Yaskawa INFORM job: A_ROOF_UPPER_0614_2_PAINT_19.JBI

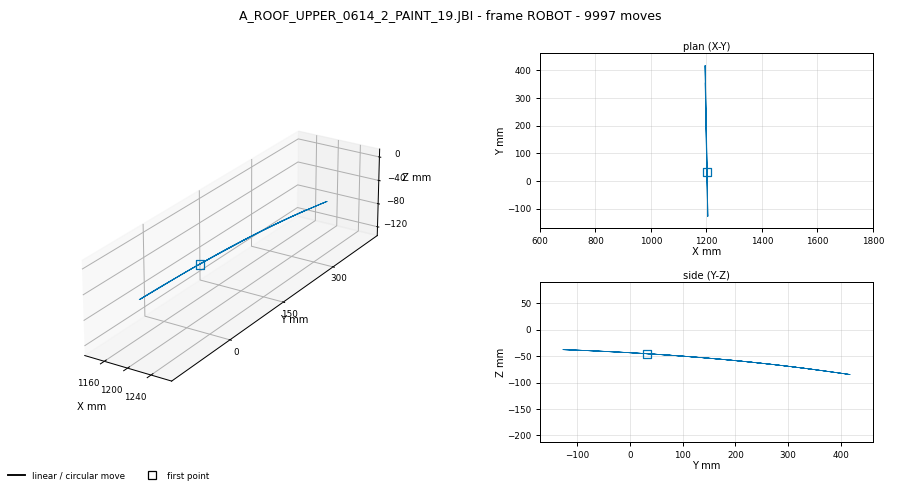
[picture p0: tool path of A_ROOF_UPPER_0614_2_PAINT_19.JBI in frame ROBOT, 9997 of 9997 moves have a stored position in this frame; points joined in program order, loops and branches not executed]
/JOB
//NAME A_ROOF_UPPER_0614_2_PAINT19
//POS
///NPOS 9997,0,0,0,0,0
///TOOL 1
///USER 0
///POSTYPE ROBOT
///RECTAN
///RCONF 1,0,0,0,0,0,0,0,0,0,0,0,0,0,0,0,0,0,0,0,0,0,0,0
C00000=1202.977,32.541,-45.099,-179.409,5.654,148.820
C00001=1202.972,32.790,-45.114,-179.406,5.654,148.820
C00002=1202.968,33.040,-45.130,-179.403,5.655,148.819
C00003=1202.962,33.290,-45.145,-179.401,5.655,148.818
C00004=1202.958,33.539,-45.160,-179.399,5.656,148.818
C00005=1202.952,33.788,-45.176,-179.396,5.657,148.817
C00006=1202.948,34.037,-45.191,-179.393,5.657,148.817
C00007=1202.943,34.287,-45.207,-179.391,5.658,148.816
C00008=1202.937,34.537,-45.222,-179.388,5.658,148.815
C00009=1202.933,34.786,-45.237,-179.386,5.659,148.815
C00010=1202.927,35.035,-45.253,-179.383,5.660,148.814
C00011=1202.923,35.285,-45.269,-179.380,5.660,148.813
C00012=1202.917,35.535,-45.285,-179.378,5.661,148.813
C00013=1202.912,35.784,-45.300,-179.376,5.661,148.812
C00014=1202.907,36.033,-45.315,-179.373,5.662,148.812
C00015=1202.902,36.283,-45.331,-179.370,5.663,148.811
C00016=1202.898,36.532,-45.347,-179.368,5.663,148.810
C00017=1202.893,36.781,-45.362,-179.365,5.664,148.810
C00018=1202.888,37.031,-45.378,-179.363,5.664,148.809
C00019=1202.882,37.281,-45.394,-179.360,5.665,148.808
C00020=1202.878,37.530,-45.409,-179.358,5.666,148.808
C00021=1202.872,37.779,-45.425,-179.355,5.666,148.807
C00022=1202.868,38.029,-45.440,-179.353,5.667,148.807
C00023=1202.862,38.279,-45.456,-179.350,5.667,148.806
C00024=1202.858,38.528,-45.471,-179.347,5.669,148.805
C00025=1202.853,38.778,-45.487,-179.344,5.669,148.805
C00026=1202.848,39.027,-45.503,-179.342,5.670,148.804
C00027=1202.842,39.276,-45.519,-179.340,5.671,148.804
C00028=1202.838,39.526,-45.534,-179.337,5.671,148.803
C00029=1202.833,39.775,-45.550,-179.334,5.672,148.802
C00030=1202.827,40.025,-45.565,-179.332,5.672,148.802
C00031=1202.823,40.274,-45.582,-179.330,5.673,148.801
C00032=1202.818,40.523,-45.598,-179.327,5.674,148.800
C00033=1202.813,40.773,-45.613,-179.324,5.674,148.800
C00034=1202.808,41.023,-45.629,-179.322,5.675,148.799
C00035=1202.803,41.272,-45.644,-179.319,5.676,148.799
C00036=1202.798,41.521,-45.661,-179.317,5.676,148.798
C00037=1202.793,41.771,-45.676,-179.314,5.677,148.797
C00038=1202.788,42.020,-45.692,-179.312,5.677,148.797
C00039=1202.783,42.269,-45.707,-179.309,5.678,148.796
C00040=1202.778,42.519,-45.724,-179.307,5.679,148.795
C00041=1202.773,42.768,-45.739,-179.304,5.679,148.795
C00042=1202.768,43.018,-45.755,-179.301,5.680,148.794
C00043=1202.763,43.267,-45.772,-179.299,5.682,148.794
C00044=1202.758,43.517,-45.787,-179.296,5.682,148.793
C00045=1202.753,43.767,-45.803,-179.293,5.683,148.792
C00046=1202.748,44.016,-45.819,-179.291,5.683,148.792
C00047=1202.743,44.265,-45.835,-179.289,5.684,148.791
C00048=1202.738,44.515,-45.850,-179.286,5.685,148.791
C00049=1202.733,44.763,-45.867,-179.283,5.685,148.790
C00050=1202.729,45.014,-45.883,-179.281,5.686,148.789
C00051=1202.723,45.263,-45.898,-179.279,5.687,148.789
C00052=1202.719,45.512,-45.915,-179.276,5.687,148.788
C00053=1202.713,45.762,-45.930,-179.273,5.688,148.787
C00054=1202.708,46.011,-45.946,-179.271,5.688,148.787
C00055=1202.703,46.261,-45.963,-179.269,5.689,148.786
C00056=1202.698,46.510,-45.978,-179.266,5.690,148.786
C00057=1202.694,46.760,-45.995,-179.263,5.691,148.785
C00058=1202.688,47.009,-46.011,-179.260,5.691,148.784
C00059=1202.683,47.259,-46.027,-179.258,5.692,148.784
C00060=1202.678,47.508,-46.043,-179.255,5.693,148.783
C00061=1202.673,47.757,-46.058,-179.253,5.693,148.783
C00062=1202.668,48.007,-46.075,-179.250,5.694,148.782
C00063=1202.663,48.256,-46.091,-179.248,5.695,148.781
C00064=1202.659,48.506,-46.107,-179.245,5.695,148.781
C00065=1202.653,48.755,-46.123,-179.243,5.696,148.780
C00066=1202.649,49.005,-46.140,-179.240,5.697,148.780
C00067=1202.643,49.254,-46.155,-179.238,5.697,148.779
C00068=1202.639,49.503,-46.172,-179.235,5.699,148.778
C00069=1202.634,49.753,-46.187,-179.232,5.699,148.778
C00070=1202.629,50.002,-46.204,-179.230,5.700,148.777
C00071=1202.624,50.252,-46.220,-179.227,5.701,148.777
C00072=1202.619,50.501,-46.236,-179.224,5.701,148.776
C00073=1202.614,50.750,-46.253,-179.222,5.702,148.775
C00074=1202.609,51.000,-46.269,-179.220,5.703,148.775
C00075=1202.604,51.249,-46.285,-179.217,5.703,148.774
C00076=1202.599,51.499,-46.301,-179.214,5.704,148.773
C00077=1202.594,51.748,-46.317,-179.212,5.705,148.773
C00078=1202.590,51.998,-46.333,-179.209,5.706,148.772
C00079=1202.584,52.247,-46.349,-179.206,5.707,148.772
C00080=1202.580,52.496,-46.366,-179.204,5.707,148.771
C00081=1202.574,52.746,-46.382,-179.202,5.708,148.771
C00082=1202.569,52.995,-46.399,-179.199,5.709,148.770
C00083=1202.565,53.245,-46.416,-179.196,5.709,148.769
C00084=1202.560,53.494,-46.431,-179.194,5.710,148.769
C00085=1202.555,53.744,-46.448,-179.192,5.711,148.768
C00086=1202.550,53.993,-46.464,-179.188,5.712,148.767
C00087=1202.545,54.243,-46.480,-179.186,5.712,148.767
C00088=1202.540,54.491,-46.496,-179.184,5.713,148.766
C00089=1202.534,54.761,-46.514,-179.181,5.714,148.766
C00090=1202.529,55.029,-46.532,-179.178,5.714,148.765
C00091=1202.524,55.297,-46.550,-179.175,5.716,148.764
C00092=1202.519,55.566,-46.567,-179.172,5.716,148.764
C00093=1202.513,55.815,-46.584,-179.170,5.717,148.763
C00094=1202.509,56.064,-46.601,-179.167,5.717,148.762
C00095=1202.504,56.315,-46.617,-179.165,5.718,148.762
C00096=1202.499,56.563,-46.633,-179.162,5.719,148.761
C00097=1202.494,56.813,-46.650,-179.159,5.720,148.761
C00098=1202.488,57.062,-46.667,-179.157,5.721,148.760
C00099=1202.484,57.312,-46.683,-179.154,5.722,148.759
C00100=1202.479,57.561,-46.699,-179.152,5.722,148.759
C00101=1202.474,57.810,-46.716,-179.150,5.723,148.758
C00102=1202.470,58.060,-46.732,-179.147,5.724,148.758
C00103=1202.464,58.309,-46.749,-179.144,5.724,148.757
C00104=1202.459,58.559,-46.765,-179.141,5.726,148.756
C00105=1202.455,58.808,-46.782,-179.139,5.726,148.756
C00106=1202.449,59.057,-46.798,-179.136,5.727,148.755
C00107=1202.444,59.307,-46.815,-179.134,5.728,148.755
C00108=1202.440,59.556,-46.832,-179.132,5.728,148.754
C00109=1202.435,59.805,-46.848,-179.129,5.729,148.753
C00110=1202.429,60.055,-46.866,-179.126,5.730,148.753
C00111=1202.424,60.304,-46.882,-179.124,5.731,148.752
C00112=1202.420,60.554,-46.898,-179.121,5.732,148.752
C00113=1202.415,60.803,-46.915,-179.118,5.732,148.751
C00114=1202.409,61.053,-46.931,-179.116,5.733,148.750
C00115=1202.405,61.302,-46.948,-179.114,5.734,148.750
C00116=1202.400,61.551,-46.965,-179.111,5.734,148.749
C00117=1202.395,61.801,-46.982,-179.108,5.736,148.749
C00118=1202.390,62.050,-46.998,-179.106,5.737,148.748
C00119=1202.386,62.300,-47.015,-179.103,5.737,148.748
C00120=1202.380,62.549,-47.032,-179.100,5.738,148.747
C00121=1202.375,62.798,-47.049,-179.098,5.739,148.746
C00122=1202.371,63.048,-47.065,-179.096,5.739,148.746
C00123=1202.366,63.297,-47.082,-179.092,5.741,148.745
C00124=1202.361,63.546,-47.099,-179.090,5.741,148.745
C00125=1202.355,63.796,-47.116,-179.088,5.742,148.744
C00126=1202.351,64.045,-47.133,-179.085,5.743,148.743
C00127=1202.346,64.294,-47.149,-179.083,5.743,148.743
C00128=1202.341,64.544,-47.166,-179.080,5.744,148.742
C00129=1202.336,64.794,-47.183,-179.077,5.745,148.742
C00130=1202.331,65.043,-47.200,-179.075,5.746,148.741
C00131=1202.326,65.292,-47.217,-179.072,5.747,148.741
C00132=1202.321,65.542,-47.233,-179.070,5.747,148.740
C00133=1202.316,65.791,-47.250,-179.067,5.748,148.739
C00134=1202.312,66.040,-47.268,-179.064,5.750,148.739
C00135=1202.306,66.289,-47.285,-179.062,5.750,148.738
C00136=1202.302,66.539,-47.301,-179.059,5.751,148.737
C00137=1202.296,66.789,-47.319,-179.057,5.752,148.737
C00138=1202.292,67.038,-47.335,-179.054,5.752,148.736
C00139=1202.287,67.287,-47.352,-179.052,5.753,148.736
C00140=1202.282,67.537,-47.369,-179.049,5.754,148.735
C00141=1202.277,67.786,-47.386,-179.046,5.755,148.735
C00142=1202.272,68.035,-47.404,-179.044,5.756,148.734
C00143=1202.268,68.285,-47.420,-179.041,5.756,148.733
C00144=1202.262,68.534,-47.437,-179.039,5.757,148.733
C00145=1202.257,68.783,-47.454,-179.036,5.758,148.732
C00146=1202.252,69.033,-47.471,-179.033,5.759,148.732
C00147=1202.248,69.282,-47.488,-179.031,5.760,148.731
C00148=1202.243,69.532,-47.506,-179.028,5.760,148.730
C00149=1202.238,69.781,-47.522,-179.026,5.761,148.730
C00150=1202.232,70.030,-47.539,-179.023,5.763,148.729
C00151=1202.228,70.279,-47.557,-179.021,5.764,148.729
C00152=1202.223,70.529,-47.574,-179.018,5.764,148.728
C00153=1202.218,70.779,-47.591,-179.015,5.765,148.728
C00154=1202.213,71.028,-47.607,-179.013,5.766,148.727
C00155=1202.208,71.277,-47.625,-179.010,5.767,148.727
C00156=1202.203,71.526,-47.642,-179.007,5.768,148.726
C00157=1202.198,71.776,-47.659,-179.005,5.768,148.725
C00158=1202.194,72.025,-47.677,-179.003,5.769,148.725
C00159=1202.189,72.275,-47.694,-178.999,5.770,148.724
C00160=1202.184,72.525,-47.711,-178.997,5.771,148.724
C00161=1202.179,72.773,-47.728,-178.995,5.772,148.723
C00162=1202.174,73.023,-47.746,-178.992,5.772,148.722
C00163=1202.169,73.272,-47.762,-178.989,5.774,148.722
C00164=1202.164,73.521,-47.780,-178.987,5.775,148.721
C00165=1202.159,73.771,-47.798,-178.984,5.775,148.721
C00166=1202.154,74.020,-47.814,-178.982,5.776,148.720
C00167=1202.150,74.270,-47.832,-178.979,5.777,148.720
C00168=1202.144,74.519,-47.849,-178.976,5.778,148.719
C00169=1202.140,74.768,-47.866,-178.974,5.779,148.718
C00170=1202.134,75.017,-47.884,-178.971,5.780,148.718
C00171=1202.130,75.266,-47.901,-178.969,5.781,148.717
C00172=1202.125,75.516,-47.918,-178.966,5.782,148.717
C00173=1202.120,75.766,-47.936,-178.963,5.782,148.716
C00174=1202.115,76.015,-47.954,-178.961,5.783,148.716
C00175=1202.110,76.265,-47.970,-178.959,5.784,148.715
C00176=1202.105,76.514,-47.988,-178.955,5.785,148.714
C00177=1202.100,76.764,-48.006,-178.953,5.786,148.714
C00178=1202.096,77.012,-48.023,-178.951,5.787,148.713
C00179=1202.090,77.261,-48.040,-178.949,5.788,148.713
C00180=1202.085,77.511,-48.058,-178.945,5.789,148.712
C00181=1202.081,77.760,-48.074,-178.943,5.790,148.711
C00182=1202.076,78.009,-48.092,-178.941,5.791,148.711
C00183=1202.071,78.259,-48.110,-178.938,5.791,148.710
C00184=1202.066,78.508,-48.128,-178.935,5.793,148.710
C00185=1202.062,78.757,-48.145,-178.933,5.793,148.709
C00186=1202.056,79.007,-48.162,-178.930,5.794,148.709
C00187=1202.052,79.256,-48.180,-178.928,5.795,148.708
C00188=1202.046,79.506,-48.198,-178.925,5.796,148.708
C00189=1202.041,79.755,-48.216,-178.922,5.797,148.707
C00190=1202.037,80.005,-48.232,-178.920,5.798,148.706
C00191=1202.032,80.254,-48.250,-178.917,5.798,148.706
C00192=1202.027,80.503,-48.268,-178.914,5.800,148.705
C00193=1202.022,80.772,-48.287,-178.912,5.801,148.705
C00194=1202.017,81.040,-48.306,-178.909,5.802,148.704
C00195=1202.011,81.308,-48.325,-178.906,5.803,148.703
C00196=1202.006,81.576,-48.344,-178.903,5.803,148.703
C00197=1202.001,81.825,-48.361,-178.901,5.805,148.702
C00198=1201.996,82.075,-48.379,-178.898,5.805,148.702
C00199=1201.991,82.324,-48.397,-178.895,5.806,148.701
C00200=1201.986,82.573,-48.415,-178.893,5.808,148.701
C00201=1201.981,82.823,-48.432,-178.890,5.808,148.700
C00202=1201.976,83.072,-48.450,-178.888,5.809,148.700
C00203=1201.972,83.321,-48.467,-178.885,5.810,148.699
C00204=1201.967,83.571,-48.485,-178.882,5.811,148.698
C00205=1201.962,83.820,-48.502,-178.880,5.812,148.698
C00206=1201.957,84.069,-48.520,-178.877,5.813,148.697
C00207=1201.952,84.319,-48.538,-178.875,5.814,148.697
C00208=1201.948,84.568,-48.557,-178.872,5.815,148.696
C00209=1201.943,84.818,-48.574,-178.869,5.816,148.695
C00210=1201.938,85.067,-48.592,-178.867,5.816,148.695
C00211=1201.933,85.317,-48.610,-178.864,5.818,148.694
C00212=1201.928,85.566,-48.628,-178.862,5.819,148.694
C00213=1201.924,85.815,-48.645,-178.859,5.819,148.693
C00214=1201.918,86.064,-48.663,-178.856,5.821,148.693
C00215=1201.913,86.314,-48.681,-178.854,5.822,148.692
C00216=1201.909,86.563,-48.699,-178.851,5.822,148.692
C00217=1201.904,86.812,-48.717,-178.849,5.824,148.691
C00218=1201.899,87.061,-48.735,-178.846,5.825,148.691
C00219=1201.894,87.310,-48.753,-178.844,5.825,148.690
C00220=1201.889,87.560,-48.771,-178.841,5.826,148.689
C00221=1201.884,87.810,-48.788,-178.838,5.827,148.689
C00222=1201.879,88.059,-48.806,-178.836,5.828,148.688
C00223=1201.874,88.308,-48.824,-178.833,5.829,148.688
C00224=1201.870,88.558,-48.842,-178.831,5.831,148.687
C00225=1201.865,88.807,-48.860,-178.828,5.831,148.687
C00226=1201.860,89.056,-48.878,-178.826,5.832,148.686
C00227=1201.855,89.305,-48.896,-178.823,5.834,148.686
C00228=1201.850,89.554,-48.914,-178.820,5.834,148.685
C00229=1201.846,89.804,-48.932,-178.818,5.835,148.685
C00230=1201.841,90.053,-48.950,-178.815,5.836,148.684
C00231=1201.836,90.302,-48.968,-178.813,5.837,148.683
C00232=1201.831,90.552,-48.986,-178.810,5.838,148.683
C00233=1201.826,90.801,-49.004,-178.807,5.840,148.682
C00234=1201.820,91.050,-49.023,-178.805,5.840,148.682
C00235=1201.815,91.299,-49.041,-178.802,5.841,148.681
C00236=1201.811,91.549,-49.059,-178.799,5.843,148.681
C00237=1201.806,91.799,-49.077,-178.797,5.843,148.680
C00238=1201.801,92.048,-49.095,-178.795,5.844,148.680
C00239=1201.796,92.297,-49.113,-178.791,5.845,148.679
C00240=1201.791,92.546,-49.131,-178.789,5.846,148.679
C00241=1201.787,92.795,-49.149,-178.787,5.847,148.678
C00242=1201.782,93.045,-49.167,-178.783,5.848,148.677
C00243=1201.777,93.294,-49.185,-178.781,5.849,148.677
C00244=1201.772,93.543,-49.205,-178.779,5.850,148.676
C00245=1201.767,93.792,-49.223,-178.776,5.852,148.676
C00246=1201.762,94.042,-49.241,-178.773,5.852,148.675
C00247=1201.758,94.291,-49.259,-178.771,5.853,148.675
C00248=1201.753,94.541,-49.277,-178.768,5.854,148.674
C00249=1201.748,94.790,-49.295,-178.766,5.855,148.674
C00250=1201.743,95.039,-49.313,-178.763,5.856,148.673
C00251=1201.738,95.289,-49.333,-178.761,5.858,148.673
C00252=1201.733,95.538,-49.351,-178.758,5.858,148.672
C00253=1201.729,95.787,-49.369,-178.755,5.859,148.671
C00254=1201.724,96.036,-49.387,-178.753,5.861,148.671
C00255=1201.719,96.286,-49.405,-178.750,5.861,148.670
C00256=1201.714,96.535,-49.424,-178.747,5.863,148.670
C00257=1201.709,96.784,-49.442,-178.745,5.863,148.669
C00258=1201.704,97.033,-49.460,-178.743,5.864,148.669
C00259=1201.700,97.283,-49.478,-178.739,5.866,148.668
C00260=1201.694,97.532,-49.498,-178.737,5.867,148.668
C00261=1201.690,97.781,-49.516,-178.735,5.867,148.667
C00262=1201.685,98.030,-49.534,-178.732,5.869,148.667
C00263=1201.680,98.280,-49.552,-178.729,5.870,148.666
C00264=1201.675,98.529,-49.571,-178.727,5.871,148.666
C00265=1201.670,98.778,-49.589,-178.724,5.872,148.665
C00266=1201.665,99.027,-49.607,-178.721,5.873,148.664
C00267=1201.661,99.277,-49.626,-178.719,5.874,148.664
C00268=1201.656,99.526,-49.645,-178.716,5.875,148.663
C00269=1201.651,99.775,-49.663,-178.714,5.876,148.663
C00270=1201.647,100.024,-49.682,-178.711,5.877,148.662
C00271=1201.641,100.274,-49.701,-178.709,5.878,148.662
C00272=1201.636,100.523,-49.719,-178.706,5.879,148.661
C00273=1201.632,100.772,-49.738,-178.703,5.880,148.661
C00274=1201.627,101.022,-49.756,-178.701,5.881,148.660
C00275=1201.622,101.270,-49.775,-178.698,5.883,148.660
C00276=1201.617,101.520,-49.793,-178.695,5.883,148.659
C00277=1201.612,101.770,-49.812,-178.693,5.884,148.659
C00278=1201.607,102.018,-49.831,-178.690,5.886,148.658
C00279=1201.603,102.268,-49.849,-178.688,5.887,148.658
C00280=1201.598,102.517,-49.868,-178.685,5.888,148.657
C00281=1201.593,102.766,-49.886,-178.683,5.889,148.656
C00282=1201.589,103.016,-49.905,-178.680,5.890,148.656
C00283=1201.583,103.265,-49.924,-178.677,5.891,148.655
C00284=1201.578,103.514,-49.942,-178.675,5.892,148.655
C00285=1201.573,103.764,-49.961,-178.672,5.894,148.654
C00286=1201.569,104.012,-49.980,-178.669,5.894,148.654
C00287=1201.564,104.262,-49.998,-178.667,5.895,148.653
C00288=1201.559,104.511,-50.018,-178.664,5.897,148.653
C00289=1201.554,104.760,-50.036,-178.662,5.898,148.652
C00290=1201.549,105.010,-50.055,-178.659,5.899,148.652
C00291=1201.545,105.259,-50.073,-178.657,5.900,148.651
C00292=1201.540,105.508,-50.092,-178.653,5.901,148.651
C00293=1201.535,105.758,-50.111,-178.651,5.902,148.650
C00294=1201.530,106.006,-50.130,-178.649,5.903,148.650
C00295=1201.526,106.256,-50.149,-178.646,5.905,148.649
C00296=1201.521,106.505,-50.167,-178.643,5.905,148.648
C00297=1201.516,106.774,-50.188,-178.641,5.907,148.648
C00298=1201.510,107.042,-50.208,-178.638,5.907,148.647
C00299=1201.505,107.310,-50.229,-178.635,5.909,148.647
C00300=1201.500,107.579,-50.249,-178.632,5.911,148.646
C00301=1201.495,107.828,-50.268,-178.629,5.911,148.646
C00302=1201.490,108.078,-50.287,-178.627,5.912,148.645
C00303=1201.485,108.327,-50.306,-178.624,5.914,148.645
C00304=1201.480,108.575,-50.325,-178.622,5.914,148.644
C00305=1201.476,108.825,-50.344,-178.619,5.916,148.644
C00306=1201.471,109.074,-50.362,-178.617,5.917,148.643
C00307=1201.466,109.324,-50.382,-178.614,5.918,148.643
C00308=1201.461,109.572,-50.401,-178.611,5.919,148.642
C00309=1201.456,109.822,-50.419,-178.608,5.921,148.642
C00310=1201.452,110.071,-50.438,-178.606,5.921,148.641
C00311=1201.447,110.321,-50.458,-178.604,5.922,148.641
C00312=1201.442,110.569,-50.477,-178.601,5.924,148.640
C00313=1201.437,110.819,-50.495,-178.598,5.924,148.639
C00314=1201.432,111.068,-50.515,-178.595,5.926,148.639
C00315=1201.428,111.317,-50.534,-178.593,5.927,148.639
C00316=1201.423,111.566,-50.553,-178.590,5.929,148.638
C00317=1201.418,111.816,-50.573,-178.588,5.929,148.638
C00318=1201.413,112.065,-50.591,-178.585,5.931,148.637
C00319=1201.408,112.315,-50.610,-178.583,5.932,148.637
C00320=1201.404,112.563,-50.629,-178.580,5.932,148.636
C00321=1201.399,112.813,-50.649,-178.577,5.934,148.636
C00322=1201.393,113.062,-50.668,-178.575,5.935,148.635
C00323=1201.389,113.311,-50.687,-178.572,5.937,148.634
C00324=1201.384,113.560,-50.706,-178.570,5.937,148.634
C00325=1201.379,113.810,-50.725,-178.567,5.939,148.633
C00326=1201.374,114.058,-50.744,-178.565,5.940,148.633
C00327=1201.370,114.308,-50.764,-178.562,5.941,148.632
C00328=1201.365,114.558,-50.783,-178.559,5.942,148.632
C00329=1201.360,114.806,-50.802,-178.556,5.944,148.631
C00330=1201.356,115.056,-50.822,-178.554,5.945,148.631
C00331=1201.350,115.305,-50.841,-178.551,5.946,148.630
C00332=1201.345,115.554,-50.861,-178.549,5.947,148.630
C00333=1201.341,115.803,-50.879,-178.546,5.948,148.629
C00334=1201.336,116.052,-50.899,-178.543,5.949,148.629
C00335=1201.331,116.302,-50.919,-178.541,5.951,148.628
C00336=1201.326,116.551,-50.938,-178.538,5.952,148.628
C00337=1201.322,116.800,-50.957,-178.535,5.953,148.627
C00338=1201.317,117.049,-50.976,-178.533,5.954,148.627
C00339=1201.312,117.298,-50.996,-178.531,5.955,148.626
C00340=1201.307,117.547,-51.015,-178.528,5.956,148.626
C00341=1201.303,117.796,-51.034,-178.525,5.957,148.625
C00342=1201.298,118.046,-51.054,-178.523,5.959,148.625
C00343=1201.293,118.295,-51.073,-178.520,5.960,148.624
C00344=1201.288,118.544,-51.093,-178.517,5.961,148.624
C00345=1201.284,118.794,-51.112,-178.515,5.962,148.623
C00346=1201.278,119.043,-51.131,-178.512,5.964,148.623
C00347=1201.274,119.292,-51.151,-178.510,5.964,148.622
C00348=1201.268,119.541,-51.170,-178.507,5.966,148.622
C00349=1201.264,119.791,-51.190,-178.505,5.967,148.621
C00350=1201.259,120.040,-51.209,-178.502,5.968,148.621
C00351=1201.255,120.288,-51.229,-178.499,5.969,148.620
C00352=1201.250,120.538,-51.249,-178.496,5.971,148.620
C00353=1201.245,120.787,-51.268,-178.494,5.972,148.619
C00354=1201.240,121.036,-51.288,-178.491,5.973,148.619
C00355=1201.235,121.286,-51.307,-178.489,5.974,148.618
C00356=1201.230,121.535,-51.327,-178.486,5.976,148.618
C00357=1201.225,121.784,-51.347,-178.483,5.977,148.617
C00358=1201.221,122.033,-51.366,-178.481,5.978,148.617
C00359=1201.216,122.282,-51.386,-178.478,5.980,148.616
C00360=1201.211,122.531,-51.405,-178.476,5.981,148.616
C00361=1201.207,122.780,-51.425,-178.473,5.982,148.616
C00362=1201.202,123.030,-51.445,-178.470,5.983,148.615
C00363=1201.197,123.279,-51.465,-178.468,5.985,148.614
C00364=1201.192,123.528,-51.484,-178.465,5.985,148.614
C00365=1201.187,123.777,-51.504,-178.462,5.987,148.613
C00366=1201.183,124.027,-51.524,-178.460,5.988,148.613
C00367=1201.177,124.276,-51.543,-178.457,5.989,148.612
C00368=1201.173,124.525,-51.563,-178.455,5.990,148.612
C00369=1201.168,124.774,-51.583,-178.452,5.992,148.612
C00370=1201.163,125.024,-51.603,-178.450,5.993,148.611
C00371=1201.158,125.272,-51.622,-178.447,5.995,148.611
C00372=1201.154,125.521,-51.642,-178.444,5.995,148.610
C00373=1201.149,125.771,-51.662,-178.442,5.997,148.610
C00374=1201.145,126.020,-51.681,-178.439,5.999,148.609
C00375=1201.140,126.269,-51.701,-178.436,5.999,148.609
C00376=1201.135,126.518,-51.721,-178.434,6.001,148.608
C00377=1201.131,126.767,-51.741,-178.431,6.002,148.608
C00378=1201.125,127.017,-51.761,-178.428,6.003,148.607
C00379=1201.120,127.266,-51.781,-178.426,6.004,148.607
C00380=1201.115,127.515,-51.801,-178.423,6.006,148.606
C00381=1201.111,127.764,-51.821,-178.421,6.007,148.606
C00382=1201.106,128.013,-51.841,-178.418,6.008,148.605
C00383=1201.101,128.263,-51.861,-178.416,6.009,148.605
C00384=1201.096,128.511,-51.881,-178.413,6.011,148.604
C00385=1201.092,128.761,-51.900,-178.410,6.012,148.604
C00386=1201.087,129.010,-51.921,-178.408,6.013,148.603
C00387=1201.083,129.259,-51.941,-178.405,6.015,148.603
C00388=1201.078,129.508,-51.961,-178.402,6.016,148.602
C00389=1201.073,129.757,-51.980,-178.400,6.017,148.602
C00390=1201.068,130.006,-52.001,-178.397,6.018,148.601
C00391=1201.064,130.255,-52.020,-178.394,6.020,148.601
C00392=1201.059,130.504,-52.041,-178.392,6.022,148.600
C00393=1201.054,130.754,-52.061,-178.389,6.022,148.600
C00394=1201.049,131.003,-52.081,-178.386,6.024,148.599
C00395=1201.044,131.252,-52.100,-178.384,6.025,148.599
C00396=1201.039,131.501,-52.121,-178.381,6.027,148.599
C00397=1201.035,131.751,-52.141,-178.379,6.027,148.598
C00398=1201.030,132.000,-52.161,-178.376,6.029,148.598
C00399=1201.025,132.249,-52.182,-178.374,6.031,148.597
C00400=1201.020,132.498,-52.202,-178.371,6.031,148.597
C00401=1201.016,132.766,-52.223,-178.368,6.033,148.596
C00402=1201.010,133.035,-52.245,-178.365,6.035,148.596
C00403=1201.005,133.303,-52.267,-178.362,6.036,148.595
C00404=1201.000,133.572,-52.288,-178.360,6.037,148.595
C00405=1200.995,133.821,-52.309,-178.357,6.039,148.594
C00406=1200.991,134.071,-52.329,-178.354,6.039,148.594
C00407=1200.985,134.320,-52.349,-178.352,6.041,148.593
C00408=1200.981,134.569,-52.370,-178.349,6.043,148.593
C00409=1200.976,134.817,-52.390,-178.346,6.043,148.592
C00410=1200.971,135.067,-52.410,-178.344,6.045,148.592
C00411=1200.966,135.316,-52.430,-178.342,6.046,148.591
C00412=1200.962,135.565,-52.451,-178.339,6.048,148.591
C00413=1200.957,135.815,-52.470,-178.336,6.049,148.590
C00414=1200.952,136.064,-52.491,-178.334,6.050,148.590
C00415=1200.947,136.313,-52.512,-178.331,6.052,148.589
C00416=1200.943,136.562,-52.532,-178.328,6.054,148.589
C00417=1200.938,136.811,-52.553,-178.326,6.055,148.589
C00418=1200.934,137.060,-52.572,-178.323,6.056,148.588
C00419=1200.928,137.310,-52.593,-178.320,6.057,148.588
C00420=1200.924,137.559,-52.614,-178.318,6.059,148.587
C00421=1200.920,137.808,-52.634,-178.315,6.060,148.587
C00422=1200.914,138.057,-52.655,-178.312,6.061,148.586
C00423=1200.910,138.306,-52.675,-178.310,6.063,148.586
C00424=1200.905,138.555,-52.695,-178.308,6.064,148.585
C00425=1200.900,138.805,-52.716,-178.305,6.065,148.585
C00426=1200.896,139.054,-52.736,-178.302,6.067,148.584
C00427=1200.891,139.302,-52.756,-178.300,6.068,148.584
C00428=1200.885,139.551,-52.777,-178.297,6.069,148.583
C00429=1200.881,139.800,-52.798,-178.294,6.071,148.583
C00430=1200.876,140.049,-52.819,-178.292,6.072,148.583
C00431=1200.871,140.298,-52.839,-178.289,6.074,148.582
C00432=1200.867,140.547,-52.859,-178.286,6.075,148.582
C00433=1200.862,140.796,-52.880,-178.284,6.076,148.581
C00434=1200.858,141.046,-52.901,-178.281,6.078,148.581
C00435=1200.853,141.295,-52.921,-178.279,6.079,148.580
C00436=1200.848,141.544,-52.942,-178.276,6.080,148.580
C00437=1200.844,141.793,-52.963,-178.273,6.082,148.579
C00438=1200.839,142.042,-52.984,-178.271,6.083,148.579
C00439=1200.834,142.291,-53.004,-178.268,6.085,148.578
C00440=1200.829,142.541,-53.025,-178.265,6.086,148.578
C00441=1200.825,142.790,-53.045,-178.263,6.087,148.578
C00442=1200.819,143.039,-53.066,-178.260,6.089,148.577
C00443=1200.815,143.288,-53.087,-178.257,6.091,148.577
C00444=1200.811,143.537,-53.107,-178.255,6.092,148.576
C00445=1200.805,143.786,-53.128,-178.252,6.093,148.576
C00446=1200.801,144.035,-53.148,-178.249,6.095,148.575
C00447=1200.796,144.284,-53.169,-178.247,6.096,148.575
C00448=1200.791,144.533,-53.190,-178.244,6.098,148.574
C00449=1200.786,144.782,-53.211,-178.242,6.098,148.574
C00450=1200.782,145.031,-53.231,-178.239,6.100,148.573
C00451=1200.777,145.280,-53.253,-178.236,6.102,148.573
C00452=1200.773,145.530,-53.274,-178.234,6.103,148.573
C00453=1200.768,145.779,-53.295,-178.231,6.104,148.572
C00454=1200.763,146.028,-53.316,-178.229,6.106,148.572
C00455=1200.758,146.277,-53.336,-178.226,6.107,148.571
C00456=1200.753,146.526,-53.357,-178.224,6.109,148.571
C00457=1200.749,146.775,-53.378,-178.221,6.110,148.570
C00458=1200.744,147.024,-53.399,-178.218,6.112,148.570
C00459=1200.739,147.273,-53.419,-178.216,6.113,148.570
C00460=1200.734,147.522,-53.440,-178.213,6.115,148.569
C00461=1200.730,147.772,-53.462,-178.210,6.116,148.569
C00462=1200.725,148.021,-53.483,-178.208,6.117,148.568
C00463=1200.720,148.270,-53.504,-178.205,6.119,148.568
C00464=1200.716,148.519,-53.524,-178.202,6.121,148.567
C00465=1200.711,148.767,-53.546,-178.200,6.121,148.567
C00466=1200.706,149.017,-53.567,-178.197,6.123,148.566
C00467=1200.701,149.266,-53.587,-178.195,6.125,148.566
C00468=1200.697,149.516,-53.608,-178.192,6.126,148.566
C00469=1200.692,149.764,-53.630,-178.189,6.127,148.565
C00470=1200.687,150.013,-53.650,-178.187,6.129,148.565
C00471=1200.682,150.262,-53.671,-178.184,6.130,148.564
C00472=1200.677,150.511,-53.693,-178.182,6.132,148.564
C00473=1200.673,150.760,-53.713,-178.179,6.133,148.563
C00474=1200.669,151.009,-53.735,-178.176,6.135,148.563
C00475=1200.664,151.259,-53.756,-178.174,6.136,148.562
C00476=1200.659,151.508,-53.777,-178.171,6.138,148.562
C00477=1200.654,151.756,-53.799,-178.168,6.139,148.562
C00478=1200.649,152.005,-53.819,-178.166,6.140,148.561
C00479=1200.646,152.254,-53.841,-178.163,6.142,148.561
C00480=1200.640,152.504,-53.862,-178.161,6.144,148.560
C00481=1200.635,152.753,-53.883,-178.158,6.145,148.560
C00482=1200.630,153.002,-53.905,-178.155,6.146,148.559
C00483=1200.627,153.251,-53.925,-178.153,6.148,148.559
C00484=1200.622,153.500,-53.947,-178.150,6.150,148.559
C00485=1200.616,153.749,-53.968,-178.148,6.151,148.558
C00486=1200.612,153.998,-53.990,-178.145,6.152,148.558
C00487=1200.607,154.247,-54.010,-178.142,6.154,148.557
C00488=1200.603,154.496,-54.032,-178.139,6.156,148.557
C00489=1200.598,154.745,-54.053,-178.137,6.157,148.556
C00490=1200.593,154.994,-54.075,-178.134,6.158,148.556
C00491=1200.588,155.244,-54.096,-178.131,6.160,148.556
C00492=1200.584,155.492,-54.117,-178.129,6.161,148.555
C00493=1200.579,155.741,-54.139,-178.127,6.163,148.555
C00494=1200.574,155.990,-54.160,-178.124,6.164,148.554
C00495=1200.570,156.240,-54.182,-178.121,6.166,148.554
C00496=1200.565,156.489,-54.203,-178.119,6.167,148.553
C00497=1200.560,156.737,-54.224,-178.116,6.169,148.553
C00498=1200.556,156.986,-54.246,-178.113,6.170,148.553
C00499=1200.551,157.236,-54.267,-178.111,6.172,148.552
C00500=1200.546,157.484,-54.289,-178.108,6.173,148.552
C00501=1200.541,157.734,-54.310,-178.106,6.175,148.551
C00502=1200.537,157.983,-54.332,-178.103,6.176,148.551
C00503=1200.532,158.232,-54.353,-178.100,6.178,148.551
C00504=1200.527,158.481,-54.374,-178.098,6.179,148.550
C00505=1200.522,158.749,-54.398,-178.095,6.181,148.550
C00506=1200.517,159.019,-54.421,-178.092,6.182,148.549
C00507=1200.512,159.288,-54.444,-178.089,6.184,148.549
C00508=1200.507,159.556,-54.468,-178.087,6.186,148.548
C00509=1200.502,159.806,-54.489,-178.084,6.187,148.548
C00510=1200.497,160.055,-54.511,-178.081,6.189,148.547
C00511=1200.493,160.304,-54.533,-178.078,6.191,148.547
C00512=1200.488,160.553,-54.555,-178.076,6.192,148.547
C00513=1200.483,160.802,-54.576,-178.073,6.194,148.546
C00514=1200.478,161.051,-54.597,-178.070,6.195,148.546
C00515=1200.474,161.300,-54.619,-178.068,6.197,148.545
C00516=1200.470,161.549,-54.640,-178.065,6.198,148.545
C00517=1200.465,161.797,-54.662,-178.063,6.200,148.545
C00518=1200.461,162.047,-54.684,-178.060,6.201,148.544
C00519=1200.456,162.296,-54.705,-178.057,6.203,148.544
C00520=1200.451,162.545,-54.727,-178.055,6.205,148.544
C00521=1200.446,162.794,-54.749,-178.052,6.206,148.543
C00522=1200.441,163.043,-54.771,-178.050,6.207,148.543
C00523=1200.437,163.292,-54.793,-178.047,6.209,148.542
C00524=1200.432,163.541,-54.815,-178.044,6.211,148.542
C00525=1200.427,163.790,-54.837,-178.042,6.212,148.541
C00526=1200.423,164.039,-54.859,-178.039,6.214,148.541
C00527=1200.418,164.289,-54.880,-178.036,6.215,148.540
C00528=1200.413,164.537,-54.902,-178.034,6.217,148.540
C00529=1200.408,164.786,-54.923,-178.031,6.219,148.540
C00530=1200.404,165.035,-54.945,-178.029,6.220,148.539
C00531=1200.399,165.284,-54.967,-178.026,6.222,148.539
C00532=1200.395,165.533,-54.989,-178.023,6.223,148.539
C00533=1200.390,165.782,-55.011,-178.021,6.225,148.538
C00534=1200.386,166.031,-55.033,-178.018,6.227,148.538
C00535=1200.381,166.280,-55.054,-178.016,6.228,148.537
C00536=1200.376,166.530,-55.077,-178.013,6.229,148.537
C00537=1200.371,166.778,-55.099,-178.010,6.231,148.536
C00538=1200.367,167.028,-55.121,-178.008,6.233,148.536
C00539=1200.362,167.276,-55.143,-178.005,6.235,148.536
C00540=1200.358,167.525,-55.165,-178.003,6.236,148.535
C00541=1200.353,167.774,-55.187,-178.000,6.238,148.535
C00542=1200.349,168.023,-55.209,-177.997,6.239,148.534
C00543=1200.343,168.272,-55.231,-177.994,6.241,148.534
C00544=1200.339,168.521,-55.253,-177.992,6.243,148.534
C00545=1200.334,168.770,-55.275,-177.989,6.244,148.533
C00546=1200.330,169.019,-55.297,-177.987,6.245,148.533
C00547=1200.325,169.268,-55.319,-177.984,6.247,148.533
C00548=1200.320,169.517,-55.341,-177.981,6.249,148.532
C00549=1200.315,169.765,-55.364,-177.979,6.251,148.532
C00550=1200.311,170.015,-55.386,-177.976,6.253,148.531
C00551=1200.306,170.263,-55.408,-177.974,6.253,148.531
C00552=1200.301,170.513,-55.430,-177.971,6.255,148.530
C00553=1200.296,170.762,-55.452,-177.968,6.257,148.530
C00554=1200.292,171.010,-55.475,-177.966,6.259,148.530
C00555=1200.287,171.259,-55.496,-177.963,6.260,148.529
C00556=1200.282,171.509,-55.519,-177.960,6.262,148.529
C00557=1200.278,171.757,-55.541,-177.958,6.263,148.529
C00558=1200.273,172.007,-55.563,-177.955,6.265,148.528
C00559=1200.269,172.255,-55.585,-177.953,6.267,148.528
C00560=1200.264,172.504,-55.608,-177.950,6.269,148.528
C00561=1200.259,172.754,-55.630,-177.947,6.270,148.527
C00562=1200.255,173.002,-55.652,-177.944,6.272,148.527
C00563=1200.250,173.251,-55.675,-177.942,6.274,148.526
C00564=1200.245,173.500,-55.696,-177.940,6.275,148.526
C00565=1200.241,173.749,-55.719,-177.937,6.276,148.526
C00566=1200.236,173.998,-55.742,-177.934,6.278,148.525
C00567=1200.231,174.247,-55.764,-177.932,6.280,148.525
C00568=1200.227,174.496,-55.786,-177.929,6.282,148.524
C00569=1200.222,174.745,-55.809,-177.926,6.284,148.524
C00570=1200.217,174.994,-55.831,-177.924,6.285,148.524
C00571=1200.213,175.243,-55.853,-177.921,6.286,148.523
C00572=1200.208,175.492,-55.876,-177.919,6.288,148.523
C00573=1200.204,175.740,-55.898,-177.916,6.290,148.522
C00574=1200.199,175.990,-55.921,-177.913,6.292,148.522
C00575=1200.194,176.239,-55.943,-177.910,6.293,148.522
C00576=1200.190,176.488,-55.966,-177.908,6.295,148.521
C00577=1200.185,176.737,-55.988,-177.905,6.297,148.521
C00578=1200.180,176.985,-56.011,-177.903,6.298,148.521
C00579=1200.175,177.235,-56.033,-177.900,6.300,148.520
C00580=1200.171,177.484,-56.056,-177.898,6.301,148.520
C00581=1200.166,177.733,-56.078,-177.895,6.303,148.519
C00582=1200.162,177.981,-56.101,-177.892,6.305,148.519
C00583=1200.158,178.231,-56.123,-177.890,6.307,148.519
C00584=1200.152,178.479,-56.146,-177.887,6.309,148.518
C00585=1200.148,178.728,-56.168,-177.884,6.311,148.518
C00586=1200.143,178.977,-56.192,-177.882,6.312,148.518
C00587=1200.139,179.225,-56.214,-177.879,6.313,148.517
C00588=1200.134,179.475,-56.237,-177.877,6.315,148.517
C00589=1200.130,179.724,-56.259,-177.874,6.317,148.517
C00590=1200.124,179.973,-56.282,-177.871,6.318,148.516
C00591=1200.120,180.221,-56.304,-177.868,6.320,148.516
C00592=1200.115,180.470,-56.328,-177.866,6.322,148.515
C00593=1200.111,180.720,-56.350,-177.863,6.324,148.515
C00594=1200.106,180.968,-56.373,-177.860,6.326,148.515
C00595=1200.101,181.218,-56.395,-177.858,6.327,148.514
C00596=1200.097,181.466,-56.418,-177.856,6.328,148.514
C00597=1200.092,181.715,-56.442,-177.853,6.330,148.513
C00598=1200.087,181.964,-56.463,-177.850,6.332,148.513
C00599=1200.083,182.213,-56.487,-177.848,6.334,148.513
C00600=1200.079,182.462,-56.509,-177.845,6.336,148.512
C00601=1200.074,182.711,-56.533,-177.842,6.337,148.512
C00602=1200.068,182.960,-56.555,-177.840,6.339,148.512
C00603=1200.064,183.209,-56.578,-177.837,6.341,148.511
C00604=1200.060,183.458,-56.601,-177.834,6.343,148.511
C00605=1200.056,183.706,-56.624,-177.832,6.345,148.511
C00606=1200.051,183.956,-56.646,-177.829,6.346,148.510
C00607=1200.045,184.204,-56.669,-177.826,6.348,148.510
C00608=1200.042,184.453,-56.692,-177.824,6.349,148.510
C00609=1200.036,184.723,-56.717,-177.821,6.352,148.509
C00610=1200.032,184.992,-56.742,-177.818,6.354,148.509
C00611=1200.026,185.262,-56.767,-177.815,6.355,148.508
C00612=1200.021,185.532,-56.792,-177.812,6.357,148.508
C00613=1200.017,185.780,-56.815,-177.810,6.359,148.508
C00614=1200.012,186.030,-56.838,-177.807,6.361,148.507
C00615=1200.008,186.279,-56.861,-177.804,6.362,148.507
C00616=1200.002,186.527,-56.884,-177.802,6.364,148.507
C00617=1199.998,186.776,-56.907,-177.799,6.366,148.506
C00618=1199.994,187.025,-56.930,-177.797,6.368,148.506
C00619=1199.989,187.274,-56.953,-177.794,6.370,148.505
C00620=1199.985,187.523,-56.976,-177.791,6.371,148.505
C00621=1199.980,187.772,-56.999,-177.789,6.373,148.505
C00622=1199.975,188.021,-57.023,-177.786,6.375,148.504
C00623=1199.970,188.269,-57.046,-177.783,6.377,148.504
C00624=1199.966,188.518,-57.068,-177.781,6.378,148.504
C00625=1199.961,188.767,-57.092,-177.778,6.380,148.503
C00626=1199.957,189.016,-57.115,-177.776,6.381,148.503
C00627=1199.952,189.265,-57.138,-177.773,6.383,148.503
C00628=1199.947,189.514,-57.162,-177.770,6.385,148.502
C00629=1199.943,189.763,-57.184,-177.768,6.387,148.502
C00630=1199.939,190.012,-57.208,-177.765,6.389,148.502
C00631=1199.933,190.260,-57.231,-177.763,6.390,148.501
C00632=1199.929,190.509,-57.254,-177.760,6.393,148.501
C00633=1199.924,190.758,-57.278,-177.758,6.394,148.501
C00634=1199.920,191.007,-57.300,-177.755,6.396,148.500
C00635=1199.916,191.256,-57.324,-177.752,6.398,148.500
C00636=1199.911,191.505,-57.348,-177.750,6.400,148.500
C00637=1199.906,191.754,-57.371,-177.747,6.402,148.499
C00638=1199.901,192.003,-57.394,-177.744,6.403,148.499
C00639=1199.897,192.252,-57.418,-177.742,6.405,148.499
C00640=1199.892,192.501,-57.441,-177.739,6.407,148.498
C00641=1199.887,192.750,-57.465,-177.736,6.409,148.498
C00642=1199.883,192.998,-57.487,-177.734,6.411,148.498
C00643=1199.879,193.247,-57.511,-177.731,6.413,148.497
C00644=1199.874,193.496,-57.535,-177.728,6.414,148.497
C00645=1199.869,193.744,-57.558,-177.726,6.416,148.497
C00646=1199.864,193.993,-57.581,-177.723,6.418,148.496
C00647=1199.860,194.242,-57.604,-177.720,6.420,148.496
C00648=1199.855,194.491,-57.629,-177.718,6.422,148.495
C00649=1199.850,194.740,-57.652,-177.715,6.423,148.495
C00650=1199.846,194.989,-57.675,-177.713,6.425,148.495
C00651=1199.841,195.238,-57.699,-177.710,6.427,148.494
C00652=1199.837,195.486,-57.723,-177.707,6.429,148.494
C00653=1199.832,195.735,-57.746,-177.705,6.431,148.494
C00654=1199.827,195.984,-57.769,-177.702,6.433,148.494
C00655=1199.823,196.233,-57.793,-177.700,6.435,148.493
C00656=1199.818,196.482,-57.817,-177.697,6.436,148.493
C00657=1199.813,196.731,-57.840,-177.694,6.438,148.493
C00658=1199.809,196.979,-57.864,-177.692,6.440,148.492
C00659=1199.804,197.228,-57.888,-177.689,6.442,148.492
C00660=1199.800,197.477,-57.911,-177.686,6.444,148.492
C00661=1199.796,197.726,-57.935,-177.684,6.446,148.491
C00662=1199.791,197.975,-57.959,-177.681,6.447,148.491
C00663=1199.787,198.224,-57.983,-177.678,6.449,148.491
C00664=1199.782,198.473,-58.006,-177.676,6.451,148.490
C00665=1199.777,198.722,-58.030,-177.673,6.453,148.490
C00666=1199.773,198.970,-58.054,-177.671,6.455,148.489
C00667=1199.768,199.219,-58.077,-177.668,6.457,148.489
C00668=1199.764,199.468,-58.101,-177.666,6.459,148.489
C00669=1199.759,199.717,-58.124,-177.663,6.460,148.489
C00670=1199.754,199.965,-58.149,-177.660,6.462,148.488
C00671=1199.749,200.214,-58.172,-177.658,6.464,148.488
C00672=1199.745,200.463,-58.197,-177.655,6.466,148.488
C00673=1199.740,200.712,-58.220,-177.652,6.468,148.487
C00674=1199.736,200.960,-58.244,-177.650,6.469,148.487
C00675=1199.732,201.210,-58.268,-177.647,6.471,148.487
C00676=1199.727,201.458,-58.292,-177.644,6.473,148.486
C00677=1199.723,201.708,-58.315,-177.642,6.475,148.486
C00678=1199.718,201.956,-58.340,-177.640,6.477,148.486
C00679=1199.713,202.205,-58.363,-177.637,6.479,148.485
C00680=1199.708,202.454,-58.387,-177.634,6.481,148.485
C00681=1199.704,202.702,-58.411,-177.632,6.483,148.485
C00682=1199.699,202.951,-58.435,-177.628,6.485,148.484
C00683=1199.696,203.200,-58.459,-177.626,6.487,148.484
C00684=1199.690,203.449,-58.484,-177.623,6.489,148.484
C00685=1199.686,203.698,-58.507,-177.621,6.491,148.483
C00686=1199.681,203.946,-58.531,-177.618,6.493,148.483
C00687=1199.677,204.195,-58.555,-177.616,6.495,148.483
C00688=1199.672,204.444,-58.579,-177.613,6.496,148.483
C00689=1199.668,204.693,-58.604,-177.610,6.498,148.482
C00690=1199.663,204.942,-58.628,-177.608,6.500,148.482
C00691=1199.659,205.191,-58.651,-177.605,6.502,148.482
C00692=1199.654,205.439,-58.676,-177.602,6.504,148.481
C00693=1199.649,205.688,-58.700,-177.600,6.506,148.481
C00694=1199.644,205.937,-58.723,-177.598,6.508,148.481
C00695=1199.641,206.186,-58.748,-177.595,6.509,148.480
C00696=1199.635,206.435,-58.772,-177.592,6.511,148.480
C00697=1199.631,206.683,-58.796,-177.590,6.513,148.480
C00698=1199.627,206.932,-58.820,-177.586,6.516,148.479
C00699=1199.621,207.181,-58.844,-177.584,6.518,148.479
C00700=1199.617,207.430,-58.869,-177.581,6.519,148.479
C00701=1199.613,207.678,-58.893,-177.579,6.522,148.479
C00702=1199.608,207.927,-58.918,-177.576,6.523,148.478
C00703=1199.604,208.176,-58.942,-177.574,6.525,148.478
C00704=1199.600,208.425,-58.966,-177.571,6.527,148.478
C00705=1199.594,208.674,-58.990,-177.568,6.529,148.477
C00706=1199.590,208.922,-59.014,-177.566,6.531,148.477
C00707=1199.585,209.171,-59.039,-177.563,6.533,148.477
C00708=1199.581,209.420,-59.063,-177.561,6.535,148.477
C00709=1199.577,209.669,-59.087,-177.558,6.537,148.476
C00710=1199.571,209.917,-59.112,-177.555,6.539,148.476
C00711=1199.567,210.166,-59.136,-177.552,6.541,148.476
C00712=1199.563,210.415,-59.161,-177.550,6.543,148.475
C00713=1199.558,210.685,-59.187,-177.547,6.545,148.475
C00714=1199.553,210.956,-59.213,-177.544,6.547,148.475
C00715=1199.548,211.226,-59.240,-177.541,6.549,148.474
C00716=1199.543,211.497,-59.267,-177.539,6.551,148.474
C00717=1199.539,211.745,-59.291,-177.536,6.553,148.474
C00718=1199.533,211.994,-59.316,-177.533,6.556,148.473
C00719=1199.530,212.243,-59.340,-177.531,6.558,148.473
C00720=1199.525,212.492,-59.365,-177.528,6.559,148.473
C00721=1199.520,212.740,-59.389,-177.525,6.561,148.472
C00722=1199.515,212.989,-59.414,-177.523,6.563,148.472
C00723=1199.511,213.238,-59.438,-177.520,6.565,148.472
C00724=1199.506,213.487,-59.463,-177.518,6.567,148.472
C00725=1199.502,213.735,-59.487,-177.515,6.569,148.471
C00726=1199.497,213.984,-59.513,-177.513,6.571,148.471
C00727=1199.493,214.233,-59.537,-177.509,6.573,148.471
C00728=1199.488,214.481,-59.561,-177.507,6.575,148.471
C00729=1199.484,214.730,-59.586,-177.504,6.577,148.470
C00730=1199.479,214.979,-59.610,-177.502,6.579,148.470
C00731=1199.474,215.229,-59.635,-177.499,6.581,148.470
C00732=1199.470,215.477,-59.660,-177.497,6.583,148.469
C00733=1199.465,215.725,-59.685,-177.494,6.585,148.469
C00734=1199.461,215.974,-59.709,-177.491,6.588,148.469
C00735=1199.456,216.223,-59.734,-177.489,6.589,148.468
C00736=1199.452,216.471,-59.758,-177.486,6.591,148.468
C00737=1199.448,216.720,-59.784,-177.483,6.593,148.468
C00738=1199.443,216.969,-59.808,-177.481,6.595,148.468
C00739=1199.439,217.218,-59.833,-177.478,6.597,148.467
C00740=1199.434,217.467,-59.858,-177.476,6.599,148.467
C00741=1199.429,217.715,-59.883,-177.473,6.602,148.467
C00742=1199.425,217.964,-59.907,-177.470,6.603,148.466
C00743=1199.420,218.213,-59.932,-177.468,6.605,148.466
C00744=1199.416,218.461,-59.958,-177.465,6.607,148.466
C00745=1199.411,218.710,-59.982,-177.462,6.609,148.466
C00746=1199.407,218.959,-60.007,-177.460,6.611,148.465
C00747=1199.402,219.207,-60.032,-177.458,6.613,148.465
C00748=1199.398,219.456,-60.057,-177.454,6.616,148.465
C00749=1199.393,219.705,-60.081,-177.452,6.618,148.465
C00750=1199.388,219.953,-60.107,-177.449,6.619,148.464
C00751=1199.384,220.202,-60.131,-177.447,6.622,148.464
C00752=1199.379,220.451,-60.156,-177.444,6.623,148.464
C00753=1199.375,220.700,-60.182,-177.442,6.625,148.463
C00754=1199.371,220.948,-60.206,-177.439,6.628,148.463
C00755=1199.366,221.197,-60.232,-177.436,6.630,148.463
C00756=1199.361,221.446,-60.256,-177.434,6.632,148.463
C00757=1199.357,221.695,-60.282,-177.431,6.634,148.462
C00758=1199.353,221.943,-60.306,-177.428,6.636,148.462
C00759=1199.348,222.192,-60.332,-177.426,6.638,148.462
C00760=1199.343,222.441,-60.356,-177.423,6.640,148.462
C00761=1199.339,222.689,-60.382,-177.420,6.642,148.461
C00762=1199.334,222.938,-60.407,-177.418,6.644,148.461
C00763=1199.330,223.187,-60.432,-177.416,6.646,148.461
C00764=1199.325,223.435,-60.457,-177.413,6.648,148.461
C00765=1199.321,223.684,-60.482,-177.410,6.650,148.460
C00766=1199.316,223.933,-60.507,-177.407,6.653,148.460
C00767=1199.312,224.182,-60.533,-177.405,6.655,148.460
C00768=1199.307,224.430,-60.558,-177.402,6.657,148.460
C00769=1199.303,224.679,-60.583,-177.400,6.658,148.459
C00770=1199.299,224.928,-60.608,-177.398,6.660,148.459
C00771=1199.294,225.176,-60.633,-177.395,6.662,148.459
C00772=1199.290,225.425,-60.659,-177.392,6.665,148.458
C00773=1199.285,225.673,-60.684,-177.389,6.667,148.458
C00774=1199.280,225.923,-60.709,-177.387,6.669,148.458
C00775=1199.275,226.171,-60.735,-177.384,6.671,148.458
C00776=1199.271,226.420,-60.760,-177.382,6.673,148.457
C00777=1199.267,226.669,-60.785,-177.379,6.676,148.457
C00778=1199.263,226.917,-60.810,-177.376,6.677,148.457
C00779=1199.258,227.166,-60.836,-177.374,6.679,148.457
C00780=1199.253,227.414,-60.861,-177.371,6.681,148.457
C00781=1199.249,227.663,-60.886,-177.369,6.683,148.456
C00782=1199.245,227.912,-60.912,-177.366,6.686,148.456
C00783=1199.240,228.160,-60.938,-177.363,6.688,148.456
C00784=1199.236,228.409,-60.963,-177.361,6.690,148.455
C00785=1199.231,228.658,-60.988,-177.358,6.692,148.455
C00786=1199.226,228.906,-61.014,-177.355,6.694,148.455
C00787=1199.222,229.155,-61.039,-177.353,6.697,148.455
C00788=1199.217,229.403,-61.065,-177.350,6.698,148.454
C00789=1199.213,229.652,-61.091,-177.347,6.700,148.454
C00790=1199.208,229.902,-61.116,-177.345,6.702,148.454
C00791=1199.204,230.150,-61.141,-177.343,6.704,148.454
C00792=1199.199,230.398,-61.167,-177.339,6.707,148.453
C00793=1199.195,230.647,-61.193,-177.337,6.709,148.453
C00794=1199.190,230.895,-61.218,-177.335,6.711,148.453
C00795=1199.186,231.144,-61.244,-177.332,6.713,148.453
C00796=1199.182,231.393,-61.269,-177.330,6.715,148.453
C00797=1199.177,231.641,-61.295,-177.327,6.718,148.452
C00798=1199.173,231.890,-61.321,-177.324,6.719,148.452
C00799=1199.168,232.139,-61.347,-177.322,6.722,148.452
C00800=1199.163,232.387,-61.372,-177.319,6.723,148.451
C00801=1199.159,232.637,-61.397,-177.316,6.726,148.451
C00802=1199.154,232.885,-61.423,-177.314,6.728,148.451
C00803=1199.150,233.133,-61.448,-177.311,6.730,148.451
C00804=1199.145,233.382,-61.474,-177.309,6.732,148.451
C00805=1199.141,233.631,-61.500,-177.306,6.735,148.450
C00806=1199.137,233.879,-61.526,-177.303,6.737,148.450
C00807=1199.132,234.127,-61.552,-177.301,6.739,148.450
C00808=1199.127,234.376,-61.578,-177.298,6.741,148.450
C00809=1199.123,234.625,-61.604,-177.296,6.743,148.449
C00810=1199.118,234.873,-61.629,-177.293,6.746,148.449
C00811=1199.114,235.122,-61.655,-177.290,6.747,148.449
C00812=1199.110,235.371,-61.681,-177.288,6.749,148.449
C00813=1199.106,235.620,-61.707,-177.286,6.751,148.448
C00814=1199.100,235.868,-61.733,-177.282,6.754,148.448
C00815=1199.096,236.117,-61.758,-177.280,6.756,148.448
C00816=1199.092,236.366,-61.784,-177.278,6.758,148.448
C00817=1199.087,236.637,-61.813,-177.274,6.761,148.448
C00818=1199.082,236.908,-61.840,-177.272,6.763,148.447
C00819=1199.077,237.180,-61.870,-177.269,6.766,148.447
C00820=1199.072,237.452,-61.898,-177.266,6.767,148.447
C00821=1199.067,237.700,-61.923,-177.263,6.770,148.447
C00822=1199.063,237.949,-61.949,-177.261,6.772,148.446
C00823=1199.058,238.197,-61.976,-177.259,6.774,148.446
C00824=1199.054,238.446,-62.002,-177.256,6.776,148.446
C00825=1199.050,238.695,-62.028,-177.253,6.779,148.446
C00826=1199.045,238.943,-62.053,-177.251,6.781,148.445
C00827=1199.040,239.191,-62.080,-177.248,6.783,148.445
C00828=1199.036,239.440,-62.106,-177.246,6.785,148.445
C00829=1199.032,239.689,-62.131,-177.243,6.788,148.445
C00830=1199.027,239.938,-62.159,-177.240,6.790,148.445
C00831=1199.023,240.186,-62.184,-177.238,6.792,148.445
C00832=1199.018,240.434,-62.210,-177.235,6.794,148.444
C00833=1199.014,240.683,-62.237,-177.232,6.796,148.444
C00834=1199.009,240.932,-62.262,-177.230,6.798,148.444
C00835=1199.005,241.181,-62.288,-177.228,6.800,148.443
C00836=1199.001,241.429,-62.315,-177.225,6.803,148.443
C00837=1198.996,241.678,-62.341,-177.222,6.805,148.443
C00838=1198.992,241.926,-62.368,-177.220,6.807,148.443
C00839=1198.987,242.174,-62.393,-177.217,6.810,148.443
C00840=1198.983,242.423,-62.419,-177.214,6.812,148.442
C00841=1198.978,242.672,-62.446,-177.212,6.814,148.442
C00842=1198.974,242.921,-62.472,-177.209,6.816,148.442
C00843=1198.969,243.169,-62.499,-177.207,6.819,148.442
C00844=1198.965,243.418,-62.525,-177.204,6.821,148.442
C00845=1198.961,243.666,-62.551,-177.202,6.823,148.442
C00846=1198.956,243.915,-62.578,-177.199,6.825,148.441
C00847=1198.952,244.163,-62.604,-177.197,6.828,148.441
C00848=1198.947,244.412,-62.630,-177.194,6.829,148.441
C00849=1198.943,244.660,-62.657,-177.192,6.832,148.441
C00850=1198.938,244.909,-62.683,-177.189,6.834,148.440
C00851=1198.934,245.157,-62.709,-177.186,6.836,148.440
C00852=1198.929,245.406,-62.736,-177.184,6.838,148.440
C00853=1198.925,245.655,-62.762,-177.181,6.841,148.440
C00854=1198.920,245.903,-62.789,-177.178,6.843,148.440
C00855=1198.916,246.152,-62.815,-177.176,6.845,148.439
C00856=1198.911,246.400,-62.842,-177.173,6.848,148.439
C00857=1198.907,246.649,-62.868,-177.171,6.850,148.439
C00858=1198.902,246.898,-62.895,-177.168,6.852,148.439
C00859=1198.898,247.146,-62.921,-177.165,6.855,148.439
C00860=1198.894,247.395,-62.948,-177.163,6.857,148.439
C00861=1198.890,247.643,-62.974,-177.160,6.859,148.438
C00862=1198.885,247.892,-63.001,-177.158,6.862,148.438
C00863=1198.880,248.140,-63.028,-177.155,6.864,148.438
C00864=1198.876,248.389,-63.054,-177.153,6.866,148.438
C00865=1198.871,248.637,-63.081,-177.150,6.868,148.437
C00866=1198.867,248.886,-63.108,-177.148,6.871,148.437
C00867=1198.863,249.135,-63.134,-177.145,6.872,148.437
C00868=1198.858,249.383,-63.161,-177.142,6.875,148.437
C00869=1198.854,249.631,-63.187,-177.140,6.877,148.437
C00870=1198.849,249.880,-63.215,-177.137,6.879,148.437
C00871=1198.845,250.128,-63.241,-177.134,6.882,148.436
C00872=1198.840,250.377,-63.267,-177.132,6.884,148.436
C00873=1198.836,250.626,-63.294,-177.129,6.886,148.436
C00874=1198.832,250.874,-63.321,-177.127,6.889,148.436
C00875=1198.827,251.122,-63.348,-177.124,6.891,148.436
C00876=1198.823,251.371,-63.375,-177.122,6.893,148.435
C00877=1198.819,251.619,-63.401,-177.119,6.896,148.435
C00878=1198.814,251.868,-63.428,-177.117,6.898,148.435
C00879=1198.809,252.117,-63.455,-177.114,6.900,148.435
C00880=1198.804,252.365,-63.482,-177.111,6.903,148.435
C00881=1198.801,252.614,-63.509,-177.109,6.905,148.435
C00882=1198.796,252.863,-63.536,-177.106,6.907,148.434
C00883=1198.792,253.111,-63.563,-177.104,6.910,148.434
C00884=1198.788,253.359,-63.589,-177.101,6.912,148.434
C00885=1198.783,253.608,-63.616,-177.098,6.915,148.434
C00886=1198.778,253.856,-63.643,-177.096,6.917,148.434
C00887=1198.774,254.105,-63.671,-177.094,6.919,148.434
C00888=1198.769,254.353,-63.698,-177.090,6.921,148.433
C00889=1198.765,254.601,-63.724,-177.088,6.924,148.433
C00890=1198.761,254.850,-63.751,-177.086,6.925,148.433
C00891=1198.757,255.099,-63.779,-177.083,6.928,148.433
C00892=1198.752,255.348,-63.806,-177.081,6.931,148.433
C00893=1198.748,255.596,-63.832,-177.078,6.933,148.432
C00894=1198.743,255.844,-63.859,-177.075,6.935,148.432
C00895=1198.739,256.093,-63.886,-177.073,6.937,148.432
C00896=1198.734,256.341,-63.913,-177.070,6.940,148.432
C00897=1198.729,256.590,-63.940,-177.068,6.942,148.432
C00898=1198.725,256.839,-63.968,-177.065,6.944,148.432
C00899=1198.721,257.087,-63.996,-177.063,6.947,148.432
C00900=1198.717,257.335,-64.022,-177.060,6.949,148.431
C00901=1198.712,257.583,-64.049,-177.057,6.952,148.431
C00902=1198.708,257.832,-64.076,-177.055,6.954,148.431
C00903=1198.703,258.080,-64.103,-177.053,6.956,148.431
C00904=1198.699,258.330,-64.131,-177.050,6.959,148.431
C00905=1198.695,258.578,-64.158,-177.047,6.961,148.430
C00906=1198.690,258.826,-64.185,-177.044,6.964,148.430
C00907=1198.685,259.075,-64.212,-177.042,6.966,148.430
C00908=1198.681,259.323,-64.240,-177.040,6.968,148.430
C00909=1198.677,259.572,-64.267,-177.037,6.971,148.430
C00910=1198.673,259.820,-64.294,-177.034,6.973,148.430
C00911=1198.668,260.068,-64.321,-177.032,6.976,148.430
C00912=1198.664,260.317,-64.348,-177.029,6.978,148.429
C00913=1198.659,260.565,-64.376,-177.026,6.981,148.429
C00914=1198.655,260.814,-64.403,-177.024,6.983,148.429
C00915=1198.651,261.062,-64.431,-177.022,6.985,148.429
C00916=1198.646,261.310,-64.458,-177.019,6.988,148.429
C00917=1198.642,261.559,-64.485,-177.016,6.990,148.429
C00918=1198.638,261.808,-64.513,-177.013,6.993,148.428
C00919=1198.633,262.056,-64.541,-177.011,6.995,148.428
C00920=1198.629,262.304,-64.568,-177.009,6.997,148.428
C00921=1198.624,262.578,-64.598,-177.006,7.000,148.428
C00922=1198.619,262.850,-64.629,-177.003,7.002,148.428
C00923=1198.614,263.123,-64.658,-177.000,7.005,148.428
C00924=1198.609,263.396,-64.689,-176.997,7.008,148.427
C00925=1198.605,263.644,-64.716,-176.995,7.010,148.427
C00926=1198.600,263.892,-64.744,-176.993,7.012,148.427
C00927=1198.596,264.141,-64.771,-176.989,7.015,148.427
C00928=1198.592,264.389,-64.799,-176.987,7.017,148.427
C00929=1198.587,264.638,-64.826,-176.984,7.020,148.427
C00930=1198.583,264.886,-64.854,-176.982,7.022,148.427
C00931=1198.578,265.135,-64.882,-176.979,7.025,148.427
C00932=1198.574,265.383,-64.910,-176.977,7.027,148.426
C00933=1198.569,265.632,-64.937,-176.974,7.030,148.426
C00934=1198.565,265.880,-64.965,-176.972,7.032,148.426
C00935=1198.561,266.129,-64.992,-176.969,7.034,148.426
C00936=1198.556,266.376,-65.020,-176.966,7.037,148.426
C00937=1198.552,266.626,-65.047,-176.964,7.039,148.426
C00938=1198.547,266.874,-65.076,-176.961,7.042,148.425
C00939=1198.543,267.122,-65.103,-176.959,7.044,148.425
C00940=1198.539,267.371,-65.131,-176.956,7.047,148.425
C00941=1198.535,267.619,-65.159,-176.954,7.049,148.425
C00942=1198.530,267.867,-65.186,-176.951,7.052,148.425
C00943=1198.525,268.116,-65.214,-176.949,7.054,148.425
C00944=1198.521,268.364,-65.242,-176.946,7.057,148.425
C00945=1198.517,268.613,-65.270,-176.943,7.059,148.425
C00946=1198.513,268.861,-65.297,-176.941,7.062,148.425
C00947=1198.508,269.109,-65.326,-176.939,7.064,148.424
C00948=1198.504,269.358,-65.354,-176.935,7.067,148.424
C00949=1198.499,269.606,-65.381,-176.933,7.069,148.424
C00950=1198.495,269.855,-65.409,-176.931,7.071,148.424
C00951=1198.490,270.103,-65.437,-176.928,7.074,148.424
C00952=1198.486,270.351,-65.465,-176.926,7.076,148.424
C00953=1198.482,270.600,-65.493,-176.923,7.079,148.424
C00954=1198.478,270.848,-65.520,-176.920,7.081,148.423
C00955=1198.473,271.097,-65.549,-176.918,7.084,148.423
C00956=1198.469,271.345,-65.577,-176.916,7.086,148.423
C00957=1198.465,271.593,-65.605,-176.913,7.089,148.423
C00958=1198.460,271.842,-65.633,-176.910,7.091,148.423
C00959=1198.455,272.090,-65.660,-176.908,7.094,148.423
C00960=1198.451,272.339,-65.689,-176.905,7.096,148.423
C00961=1198.446,272.587,-65.717,-176.902,7.099,148.423
C00962=1198.443,272.835,-65.745,-176.900,7.101,148.422
C00963=1198.438,273.083,-65.773,-176.897,7.104,148.422
C00964=1198.434,273.332,-65.802,-176.895,7.106,148.422
C00965=1198.429,273.580,-65.829,-176.892,7.109,148.422
C00966=1198.425,273.829,-65.858,-176.890,7.111,148.422
C00967=1198.421,274.077,-65.886,-176.887,7.114,148.422
C00968=1198.417,274.325,-65.914,-176.885,7.116,148.422
C00969=1198.412,274.574,-65.942,-176.882,7.119,148.422
C00970=1198.408,274.822,-65.971,-176.880,7.121,148.422
C00971=1198.403,275.070,-65.999,-176.877,7.124,148.422
C00972=1198.399,275.319,-66.027,-176.875,7.126,148.421
C00973=1198.394,275.567,-66.056,-176.872,7.129,148.421
C00974=1198.390,275.816,-66.084,-176.869,7.132,148.421
C00975=1198.386,276.064,-66.111,-176.867,7.134,148.421
C00976=1198.381,276.313,-66.140,-176.864,7.137,148.421
C00977=1198.377,276.560,-66.168,-176.862,7.139,148.421
C00978=1198.373,276.809,-66.197,-176.859,7.142,148.421
C00979=1198.368,277.057,-66.224,-176.857,7.144,148.421
C00980=1198.364,277.306,-66.253,-176.854,7.147,148.421
C00981=1198.360,277.555,-66.281,-176.851,7.149,148.420
C00982=1198.355,277.803,-66.310,-176.849,7.152,148.420
C00983=1198.352,278.051,-66.339,-176.847,7.154,148.420
C00984=1198.346,278.299,-66.367,-176.844,7.157,148.420
C00985=1198.343,278.548,-66.395,-176.842,7.159,148.420
C00986=1198.338,278.796,-66.423,-176.839,7.162,148.420
C00987=1198.333,279.045,-66.452,-176.836,7.164,148.420
C00988=1198.330,279.293,-66.481,-176.834,7.167,148.420
C00989=1198.325,279.541,-66.509,-176.831,7.170,148.420
C00990=1198.321,279.789,-66.538,-176.829,7.172,148.420
C00991=1198.316,280.038,-66.566,-176.826,7.175,148.419
C00992=1198.312,280.286,-66.594,-176.823,7.177,148.419
C00993=1198.308,280.534,-66.624,-176.821,7.180,148.419
C00994=1198.303,280.783,-66.652,-176.819,7.183,148.419
C00995=1198.299,281.031,-66.680,-176.816,7.186,148.419
C00996=1198.295,281.279,-66.709,-176.813,7.187,148.419
C00997=1198.290,281.528,-66.738,-176.811,7.190,148.419
C00998=1198.286,281.776,-66.766,-176.808,7.193,148.419
C00999=1198.282,282.024,-66.795,-176.806,7.196,148.419
C01000=1198.277,282.273,-66.824,-176.803,7.199,148.419
C01001=1198.273,282.521,-66.852,-176.800,7.200,148.418
C01002=1198.268,282.769,-66.881,-176.798,7.203,148.418
C01003=1198.264,283.018,-66.910,-176.796,7.206,148.418
C01004=1198.260,283.266,-66.939,-176.793,7.209,148.418
C01005=1198.255,283.514,-66.967,-176.791,7.211,148.418
C01006=1198.251,283.763,-66.996,-176.788,7.214,148.418
C01007=1198.247,284.011,-67.025,-176.785,7.217,148.418
C01008=1198.243,284.260,-67.053,-176.783,7.219,148.418
C01009=1198.238,284.507,-67.082,-176.780,7.222,148.418
C01010=1198.233,284.756,-67.111,-176.778,7.224,148.418
C01011=1198.230,285.004,-67.140,-176.775,7.227,148.418
C01012=1198.225,285.252,-67.168,-176.773,7.229,148.418
C01013=1198.221,285.500,-67.198,-176.770,7.232,148.418
C01014=1198.216,285.749,-67.227,-176.767,7.235,148.417
C01015=1198.212,285.997,-67.255,-176.765,7.237,148.417
C01016=1198.208,286.245,-67.284,-176.762,7.240,148.417
C01017=1198.204,286.494,-67.313,-176.760,7.242,148.417
C01018=1198.199,286.742,-67.343,-176.757,7.245,148.417
C01019=1198.194,286.990,-67.371,-176.755,7.248,148.417
C01020=1198.190,287.238,-67.401,-176.753,7.250,148.417
C01021=1198.186,287.487,-67.429,-176.750,7.253,148.417
C01022=1198.182,287.735,-67.458,-176.747,7.255,148.417
C01023=1198.177,287.983,-67.487,-176.745,7.258,148.417
C01024=1198.173,288.232,-67.516,-176.742,7.261,148.417
C01025=1198.168,288.505,-67.548,-176.739,7.264,148.417
C01026=1198.164,288.780,-67.580,-176.737,7.267,148.417
C01027=1198.159,289.055,-67.613,-176.734,7.269,148.417
C01028=1198.154,289.329,-67.645,-176.731,7.272,148.416
C01029=1198.150,289.578,-67.674,-176.729,7.275,148.416
C01030=1198.145,289.826,-67.703,-176.726,7.278,148.416
C01031=1198.141,290.074,-67.732,-176.724,7.280,148.416
C01032=1198.137,290.322,-67.762,-176.721,7.283,148.416
C01033=1198.132,290.571,-67.790,-176.718,7.286,148.416
C01034=1198.128,290.819,-67.820,-176.716,7.289,148.416
C01035=1198.124,291.067,-67.849,-176.713,7.292,148.416
C01036=1198.120,291.315,-67.878,-176.711,7.294,148.416
C01037=1198.115,291.563,-67.907,-176.709,7.297,148.416
C01038=1198.111,291.812,-67.936,-176.706,7.300,148.416
C01039=1198.107,292.060,-67.965,-176.704,7.302,148.416
C01040=1198.103,292.308,-67.995,-176.701,7.305,148.416
C01041=1198.098,292.557,-68.024,-176.698,7.307,148.416
C01042=1198.094,292.805,-68.054,-176.696,7.310,148.416
C01043=1198.090,293.053,-68.083,-176.693,7.313,148.416
C01044=1198.085,293.301,-68.112,-176.691,7.315,148.415
C01045=1198.081,293.549,-68.142,-176.688,7.318,148.415
C01046=1198.077,293.797,-68.171,-176.685,7.321,148.415
C01047=1198.072,294.046,-68.200,-176.683,7.323,148.415
C01048=1198.068,294.294,-68.229,-176.681,7.326,148.415
C01049=1198.063,294.543,-68.260,-176.678,7.329,148.415
C01050=1198.059,294.791,-68.289,-176.676,7.332,148.415
C01051=1198.055,295.039,-68.318,-176.673,7.335,148.415
C01052=1198.051,295.288,-68.348,-176.671,7.337,148.415
C01053=1198.046,295.535,-68.377,-176.668,7.340,148.415
C01054=1198.042,295.784,-68.406,-176.666,7.343,148.415
C01055=1198.038,296.032,-68.436,-176.663,7.345,148.415
C01056=1198.034,296.279,-68.466,-176.661,7.348,148.415
C01057=1198.030,296.528,-68.495,-176.658,7.351,148.415
C01058=1198.025,296.776,-68.525,-176.656,7.353,148.415
C01059=1198.021,297.024,-68.554,-176.653,7.356,148.415
C01060=1198.016,297.273,-68.584,-176.650,7.359,148.415
C01061=1198.012,297.521,-68.614,-176.648,7.361,148.415
C01062=1198.008,297.769,-68.643,-176.646,7.364,148.415
C01063=1198.004,298.018,-68.673,-176.644,7.367,148.415
C01064=1198.000,298.266,-68.702,-176.641,7.370,148.415
C01065=1197.996,298.514,-68.732,-176.638,7.373,148.415
C01066=1197.991,298.762,-68.762,-176.636,7.375,148.415
C01067=1197.987,299.010,-68.792,-176.633,7.378,148.415
C01068=1197.982,299.259,-68.821,-176.631,7.381,148.415
C01069=1197.978,299.507,-68.851,-176.628,7.383,148.415
C01070=1197.974,299.755,-68.882,-176.626,7.386,148.415
C01071=1197.969,300.003,-68.911,-176.623,7.389,148.415
C01072=1197.965,300.251,-68.941,-176.621,7.391,148.414
C01073=1197.961,300.500,-68.970,-176.618,7.394,148.414
C01074=1197.956,300.748,-69.001,-176.616,7.397,148.414
C01075=1197.952,300.996,-69.030,-176.613,7.399,148.414
C01076=1197.948,301.244,-69.060,-176.611,7.402,148.414
C01077=1197.944,301.492,-69.090,-176.608,7.405,148.414
C01078=1197.939,301.740,-69.120,-176.606,7.408,148.414
C01079=1197.935,301.989,-69.149,-176.603,7.411,148.414
C01080=1197.931,302.236,-69.179,-176.601,7.414,148.414
C01081=1197.926,302.485,-69.210,-176.599,7.416,148.414
C01082=1197.922,302.733,-69.239,-176.596,7.419,148.414
C01083=1197.918,302.981,-69.269,-176.593,7.422,148.414
C01084=1197.913,303.229,-69.299,-176.591,7.424,148.414
C01085=1197.909,303.477,-69.329,-176.589,7.427,148.414
C01086=1197.905,303.725,-69.359,-176.586,7.430,148.414
C01087=1197.901,303.973,-69.390,-176.584,7.433,148.414
C01088=1197.896,304.222,-69.419,-176.581,7.436,148.414
C01089=1197.892,304.470,-69.448,-176.578,7.439,148.414
C01090=1197.888,304.718,-69.479,-176.576,7.442,148.414
C01091=1197.884,304.967,-69.509,-176.573,7.444,148.414
C01092=1197.879,305.215,-69.540,-176.571,7.447,148.414
C01093=1197.875,305.463,-69.569,-176.569,7.450,148.414
C01094=1197.871,305.711,-69.600,-176.566,7.452,148.414
C01095=1197.867,305.959,-69.630,-176.564,7.455,148.414
C01096=1197.863,306.207,-69.660,-176.561,7.458,148.414
C01097=1197.858,306.455,-69.690,-176.559,7.461,148.414
C01098=1197.854,306.703,-69.720,-176.556,7.464,148.414
C01099=1197.849,306.951,-69.751,-176.553,7.467,148.414
C01100=1197.846,307.200,-69.780,-176.552,7.469,148.414
C01101=1197.841,307.448,-69.811,-176.549,7.472,148.414
C01102=1197.837,307.696,-69.841,-176.546,7.475,148.414
C01103=1197.832,307.944,-69.871,-176.544,7.477,148.414
C01104=1197.828,308.192,-69.902,-176.542,7.480,148.414
C01105=1197.824,308.440,-69.932,-176.539,7.483,148.414
C01106=1197.820,308.688,-69.962,-176.536,7.486,148.414
C01107=1197.816,308.937,-69.993,-176.535,7.489,148.414
C01108=1197.812,309.184,-70.023,-176.532,7.492,148.414
C01109=1197.807,309.433,-70.053,-176.529,7.495,148.414
C01110=1197.803,309.681,-70.083,-176.527,7.497,148.414
C01111=1197.798,309.929,-70.114,-176.524,7.500,148.414
C01112=1197.794,310.177,-70.145,-176.522,7.503,148.414
C01113=1197.790,310.425,-70.175,-176.520,7.506,148.414
C01114=1197.785,310.673,-70.205,-176.517,7.509,148.414
C01115=1197.782,310.921,-70.236,-176.515,7.512,148.414
C01116=1197.777,311.169,-70.266,-176.512,7.515,148.414
C01117=1197.773,311.418,-70.298,-176.510,7.517,148.414
C01118=1197.769,311.665,-70.328,-176.507,7.520,148.414
C01119=1197.764,311.914,-70.358,-176.505,7.523,148.414
C01120=1197.760,312.162,-70.388,-176.503,7.525,148.414
C01121=1197.756,312.409,-70.419,-176.500,7.528,148.414
C01122=1197.752,312.658,-70.450,-176.498,7.532,148.415
C01123=1197.748,312.906,-70.480,-176.495,7.535,148.415
C01124=1197.743,313.154,-70.511,-176.493,7.537,148.415
C01125=1197.739,313.402,-70.542,-176.490,7.540,148.415
C01126=1197.735,313.650,-70.572,-176.488,7.543,148.415
C01127=1197.731,313.898,-70.603,-176.486,7.546,148.415
C01128=1197.726,314.146,-70.634,-176.483,7.549,148.415
C01129=1197.722,314.423,-70.667,-176.480,7.552,148.415
C01130=1197.717,314.699,-70.702,-176.478,7.555,148.415
C01131=1197.712,314.975,-70.735,-176.475,7.559,148.415
C01132=1197.708,315.252,-70.770,-176.472,7.562,148.415
C01133=1197.703,315.500,-70.801,-176.470,7.564,148.415
C01134=1197.698,315.748,-70.832,-176.467,7.567,148.415
C01135=1197.695,315.996,-70.862,-176.465,7.570,148.415
C01136=1197.690,316.244,-70.893,-176.463,7.573,148.415
C01137=1197.686,316.492,-70.924,-176.460,7.576,148.415
C01138=1197.682,316.741,-70.955,-176.458,7.579,148.415
C01139=1197.678,316.988,-70.986,-176.455,7.582,148.415
C01140=1197.674,317.236,-71.016,-176.453,7.585,148.415
C01141=1197.670,317.484,-71.047,-176.451,7.587,148.415
C01142=1197.665,317.732,-71.078,-176.448,7.590,148.415
C01143=1197.660,317.980,-71.109,-176.446,7.593,148.415
C01144=1197.657,318.229,-71.140,-176.444,7.596,148.415
C01145=1197.652,318.477,-71.170,-176.441,7.599,148.415
C01146=1197.648,318.724,-71.202,-176.439,7.602,148.415
C01147=1197.644,318.973,-71.233,-176.436,7.605,148.415
C01148=1197.640,319.220,-71.264,-176.434,7.608,148.416
C01149=1197.636,319.469,-71.295,-176.432,7.611,148.416
C01150=1197.631,319.716,-71.326,-176.429,7.614,148.416
C01151=1197.627,319.964,-71.356,-176.427,7.617,148.416
C01152=1197.623,320.213,-71.388,-176.425,7.619,148.416
C01153=1197.619,320.461,-71.418,-176.422,7.622,148.416
C01154=1197.615,320.709,-71.450,-176.420,7.625,148.416
C01155=1197.610,320.957,-71.481,-176.417,7.628,148.416
C01156=1197.606,321.205,-71.512,-176.415,7.631,148.416
C01157=1197.602,321.453,-71.544,-176.413,7.634,148.416
C01158=1197.597,321.701,-71.574,-176.410,7.637,148.416
C01159=1197.593,321.949,-71.605,-176.408,7.640,148.416
C01160=1197.589,322.197,-71.637,-176.405,7.643,148.416
C01161=1197.585,322.445,-71.668,-176.403,7.646,148.416
C01162=1197.581,322.693,-71.699,-176.401,7.649,148.417
C01163=1197.576,322.941,-71.730,-176.398,7.651,148.416
C01164=1197.572,323.189,-71.761,-176.396,7.654,148.417
C01165=1197.569,323.436,-71.792,-176.394,7.657,148.417
C01166=1197.565,323.685,-71.823,-176.391,7.661,148.417
C01167=1197.560,323.932,-71.855,-176.389,7.663,148.417
C01168=1197.556,324.181,-71.886,-176.386,7.666,148.417
C01169=1197.551,324.429,-71.918,-176.384,7.669,148.417
C01170=1197.547,324.677,-71.949,-176.382,7.672,148.417
C01171=1197.543,324.925,-71.981,-176.380,7.675,148.417
C01172=1197.539,325.173,-72.012,-176.377,7.678,148.417
C01173=1197.535,325.421,-72.043,-176.375,7.681,148.417
C01174=1197.531,325.669,-72.074,-176.372,7.684,148.417
C01175=1197.526,325.917,-72.106,-176.371,7.687,148.418
C01176=1197.522,326.165,-72.137,-176.368,7.690,148.418
C01177=1197.518,326.413,-72.169,-176.366,7.693,148.418
C01178=1197.514,326.661,-72.200,-176.363,7.696,148.418
C01179=1197.510,326.909,-72.231,-176.361,7.699,148.418
C01180=1197.506,327.157,-72.263,-176.359,7.702,148.418
C01181=1197.501,327.405,-72.294,-176.356,7.705,148.418
C01182=1197.497,327.653,-72.326,-176.354,7.708,148.418
C01183=1197.493,327.900,-72.358,-176.352,7.710,148.418
C01184=1197.489,328.149,-72.389,-176.349,7.714,148.418
C01185=1197.484,328.396,-72.420,-176.347,7.717,148.419
C01186=1197.481,328.644,-72.452,-176.344,7.720,148.419
C01187=1197.477,328.893,-72.483,-176.343,7.722,148.419
C01188=1197.472,329.140,-72.515,-176.340,7.725,148.419
C01189=1197.468,329.389,-72.547,-176.338,7.729,148.419
C01190=1197.463,329.637,-72.578,-176.335,7.732,148.419
C01191=1197.459,329.885,-72.610,-176.333,7.734,148.419
C01192=1197.455,330.132,-72.641,-176.331,7.737,148.419
C01193=1197.451,330.380,-72.673,-176.329,7.741,148.419
C01194=1197.447,330.628,-72.706,-176.326,7.744,148.420
C01195=1197.442,330.876,-72.736,-176.324,7.746,148.419
C01196=1197.439,331.124,-72.768,-176.322,7.749,148.420
C01197=1197.434,331.372,-72.800,-176.319,7.752,148.420
C01198=1197.430,331.620,-72.832,-176.317,7.756,148.420
C01199=1197.426,331.868,-72.864,-176.315,7.758,148.420
C01200=1197.422,332.115,-72.895,-176.313,7.761,148.420
C01201=1197.418,332.364,-72.927,-176.310,7.765,148.420
C01202=1197.413,332.612,-72.959,-176.308,7.768,148.420
C01203=1197.409,332.860,-72.991,-176.306,7.770,148.420
C01204=1197.405,333.108,-73.022,-176.304,7.774,148.421
C01205=1197.400,333.355,-73.054,-176.301,7.777,148.421
C01206=1197.397,333.604,-73.086,-176.299,7.780,148.421
C01207=1197.393,333.852,-73.118,-176.297,7.782,148.421
C01208=1197.388,334.099,-73.150,-176.295,7.785,148.421
C01209=1197.384,334.347,-73.182,-176.292,7.789,148.421
C01210=1197.381,334.595,-73.214,-176.290,7.792,148.422
C01211=1197.376,334.843,-73.246,-176.288,7.794,148.421
C01212=1197.372,335.091,-73.278,-176.286,7.798,148.422
C01213=1197.368,335.339,-73.310,-176.283,7.801,148.422
C01214=1197.363,335.587,-73.342,-176.281,7.804,148.422
C01215=1197.359,335.835,-73.374,-176.279,7.806,148.422
C01216=1197.355,336.083,-73.406,-176.277,7.810,148.422
C01217=1197.351,336.330,-73.437,-176.275,7.813,148.423
C01218=1197.347,336.578,-73.469,-176.272,7.816,148.423
C01219=1197.342,336.827,-73.502,-176.270,7.819,148.423
C01220=1197.339,337.075,-73.534,-176.268,7.822,148.423
C01221=1197.334,337.322,-73.566,-176.266,7.825,148.423
C01222=1197.330,337.570,-73.598,-176.263,7.828,148.423
C01223=1197.326,337.818,-73.631,-176.261,7.831,148.423
C01224=1197.322,338.066,-73.662,-176.259,7.834,148.424
C01225=1197.317,338.314,-73.695,-176.257,7.838,148.424
C01226=1197.313,338.562,-73.726,-176.254,7.841,148.424
C01227=1197.310,338.809,-73.759,-176.253,7.843,148.424
C01228=1197.305,339.057,-73.791,-176.250,7.846,148.424
C01229=1197.301,339.305,-73.823,-176.248,7.850,148.424
C01230=1197.297,339.553,-73.855,-176.246,7.853,148.425
C01231=1197.293,339.801,-73.887,-176.243,7.856,148.425
C01232=1197.289,340.049,-73.920,-176.242,7.859,148.425
C01233=1197.284,340.327,-73.957,-176.239,7.862,148.425
C01234=1197.279,340.606,-73.992,-176.237,7.866,148.425
C01235=1197.275,340.885,-74.029,-176.234,7.869,148.425
C01236=1197.270,341.163,-74.065,-176.232,7.873,148.426
C01237=1197.266,341.411,-74.097,-176.229,7.876,148.426
C01238=1197.262,341.658,-74.130,-176.227,7.879,148.426
C01239=1197.257,341.907,-74.163,-176.226,7.882,148.426
C01240=1197.254,342.155,-74.194,-176.223,7.885,148.426
C01241=1197.249,342.402,-74.227,-176.221,7.888,148.427
C01242=1197.245,342.650,-74.259,-176.219,7.892,148.427
C01243=1197.241,342.898,-74.292,-176.217,7.894,148.427
C01244=1197.237,343.146,-74.325,-176.215,7.897,148.427
C01245=1197.233,343.394,-74.357,-176.213,7.901,148.427
C01246=1197.228,343.641,-74.389,-176.210,7.904,148.428
C01247=1197.224,343.889,-74.422,-176.208,7.906,148.428
C01248=1197.220,344.137,-74.454,-176.206,7.910,148.428
C01249=1197.216,344.385,-74.487,-176.204,7.913,148.428
C01250=1197.211,344.633,-74.519,-176.202,7.916,148.428
C01251=1197.208,344.881,-74.552,-176.200,7.919,148.428
C01252=1197.203,345.129,-74.584,-176.198,7.922,148.429
C01253=1197.199,345.376,-74.617,-176.196,7.925,148.429
C01254=1197.195,345.624,-74.650,-176.193,7.929,148.429
C01255=1197.191,345.872,-74.682,-176.192,7.931,148.429
C01256=1197.187,346.120,-74.715,-176.189,7.935,148.429
C01257=1197.182,346.368,-74.748,-176.187,7.938,148.430
C01258=1197.179,346.616,-74.780,-176.185,7.941,148.430
C01259=1197.175,346.864,-74.813,-176.183,7.944,148.430
C01260=1197.170,347.112,-74.846,-176.181,7.947,148.430
C01261=1197.166,347.359,-74.879,-176.179,7.950,148.431
C01262=1197.162,347.607,-74.910,-176.177,7.954,148.431
C01263=1197.158,347.854,-74.944,-176.175,7.957,148.431
C01264=1197.153,348.103,-74.976,-176.173,7.960,148.431
C01265=1197.149,348.350,-75.009,-176.171,7.963,148.432
C01266=1197.146,348.598,-75.042,-176.169,7.967,148.432
C01267=1197.142,348.846,-75.075,-176.167,7.969,148.432
C01268=1197.137,349.094,-75.107,-176.165,7.972,148.432
C01269=1197.133,349.342,-75.140,-176.163,7.976,148.432
C01270=1197.129,349.589,-75.174,-176.160,7.979,148.433
C01271=1197.125,349.837,-75.205,-176.159,7.982,148.433
C01272=1197.121,350.085,-75.239,-176.156,7.985,148.433
C01273=1197.117,350.333,-75.272,-176.155,7.989,148.433
C01274=1197.112,350.580,-75.305,-176.152,7.992,148.434
C01275=1197.108,350.828,-75.337,-176.151,7.994,148.434
C01276=1197.104,351.076,-75.370,-176.148,7.998,148.434
C01277=1197.100,351.324,-75.403,-176.146,8.001,148.434
C01278=1197.096,351.571,-75.436,-176.144,8.005,148.435
C01279=1197.092,351.819,-75.469,-176.143,8.007,148.435
C01280=1197.088,352.067,-75.502,-176.141,8.011,148.435
C01281=1197.083,352.315,-75.535,-176.138,8.014,148.435
C01282=1197.079,352.563,-75.568,-176.136,8.017,148.436
C01283=1197.075,352.810,-75.601,-176.135,8.020,148.436
C01284=1197.071,353.058,-75.634,-176.133,8.023,148.436
C01285=1197.067,353.306,-75.667,-176.130,8.027,148.436
C01286=1197.063,353.554,-75.700,-176.129,8.029,148.437
C01287=1197.059,353.801,-75.734,-176.127,8.033,148.437
C01288=1197.054,354.049,-75.767,-176.125,8.036,148.437
C01289=1197.050,354.297,-75.800,-176.122,8.039,148.438
C01290=1197.046,354.545,-75.833,-176.121,8.042,148.438
C01291=1197.042,354.792,-75.866,-176.119,8.046,148.438
C01292=1197.039,355.041,-75.900,-176.117,8.049,148.438
C01293=1197.034,355.288,-75.933,-176.115,8.053,148.439
C01294=1197.030,355.536,-75.966,-176.113,8.055,148.439
C01295=1197.026,355.784,-75.999,-176.111,8.058,148.439
C01296=1197.022,356.032,-76.032,-176.109,8.062,148.440
C01297=1197.018,356.279,-76.066,-176.107,8.065,148.440
C01298=1197.014,356.527,-76.099,-176.105,8.068,148.440
C01299=1197.010,356.775,-76.132,-176.104,8.072,148.440
C01300=1197.005,357.023,-76.165,-176.101,8.075,148.441
C01301=1197.001,357.270,-76.198,-176.100,8.077,148.441
C01302=1196.997,357.518,-76.231,-176.098,8.081,148.441
C01303=1196.993,357.766,-76.264,-176.096,8.084,148.442
C01304=1196.989,358.013,-76.298,-176.094,8.088,148.442
C01305=1196.985,358.261,-76.331,-176.092,8.090,148.442
C01306=1196.982,358.509,-76.365,-176.091,8.094,148.443
C01307=1196.977,358.757,-76.398,-176.088,8.097,148.443
C01308=1196.973,359.004,-76.431,-176.087,8.100,148.443
C01309=1196.969,359.252,-76.464,-176.085,8.104,148.443
C01310=1196.965,359.500,-76.498,-176.083,8.107,148.444
C01311=1196.960,359.747,-76.532,-176.081,8.111,148.444
C01312=1196.956,359.995,-76.565,-176.080,8.113,148.444
C01313=1196.952,360.243,-76.598,-176.077,8.117,148.445
C01314=1196.949,360.491,-76.632,-176.076,8.120,148.445
C01315=1196.945,360.738,-76.666,-176.074,8.123,148.445
C01316=1196.941,360.986,-76.699,-176.072,8.126,148.446
C01317=1196.936,361.234,-76.732,-176.070,8.130,148.446
C01318=1196.932,361.482,-76.766,-176.069,8.133,148.446
C01319=1196.928,361.729,-76.800,-176.067,8.136,148.447
C01320=1196.924,361.977,-76.833,-176.065,8.140,148.447
C01321=1196.920,362.225,-76.866,-176.063,8.142,148.447
C01322=1196.916,362.472,-76.900,-176.062,8.146,148.448
C01323=1196.912,362.720,-76.933,-176.060,8.149,148.448
C01324=1196.907,362.968,-76.967,-176.058,8.152,148.448
C01325=1196.903,363.215,-77.001,-176.056,8.156,148.449
C01326=1196.900,363.464,-77.035,-176.055,8.159,148.449
C01327=1196.896,363.711,-77.068,-176.053,8.162,148.450
C01328=1196.891,363.959,-77.102,-176.051,8.166,148.450
C01329=1196.887,364.206,-77.135,-176.050,8.168,148.450
C01330=1196.883,364.453,-77.169,-176.048,8.172,148.451
C01331=1196.880,364.702,-77.203,-176.046,8.174,148.451
C01332=1196.876,364.949,-77.237,-176.045,8.178,148.451
C01333=1196.871,365.197,-77.270,-176.043,8.181,148.452
C01334=1196.867,365.444,-77.304,-176.042,8.185,148.452
C01335=1196.864,365.693,-77.338,-176.040,8.188,148.453
C01336=1196.859,365.940,-77.372,-176.038,8.191,148.453
C01337=1196.855,366.221,-77.409,-176.036,8.194,148.453
C01338=1196.850,366.502,-77.448,-176.035,8.198,148.454
C01339=1196.845,366.782,-77.486,-176.033,8.202,148.454
C01340=1196.841,367.064,-77.525,-176.031,8.205,148.455
C01341=1196.837,367.311,-77.558,-176.029,8.209,148.455
C01342=1196.832,367.559,-77.593,-176.028,8.212,148.455
C01343=1196.828,367.806,-77.626,-176.026,8.215,148.456
C01344=1196.825,368.054,-77.660,-176.025,8.218,148.456
C01345=1196.820,368.302,-77.695,-176.023,8.222,148.457
C01346=1196.816,368.549,-77.728,-176.022,8.225,148.457
C01347=1196.812,368.797,-77.762,-176.020,8.228,148.458
C01348=1196.808,369.045,-77.796,-176.019,8.231,148.458
C01349=1196.804,369.292,-77.830,-176.017,8.235,148.458
C01350=1196.800,369.540,-77.864,-176.016,8.237,148.459
C01351=1196.796,369.788,-77.898,-176.014,8.241,148.459
C01352=1196.792,370.036,-77.932,-176.013,8.244,148.460
C01353=1196.788,370.283,-77.966,-176.011,8.247,148.460
C01354=1196.784,370.530,-77.999,-176.010,8.250,148.460
C01355=1196.780,370.779,-78.034,-176.009,8.253,148.461
C01356=1196.776,371.026,-78.068,-176.008,8.257,148.461
C01357=1196.771,371.274,-78.102,-176.006,8.260,148.462
C01358=1196.768,371.521,-78.136,-176.004,8.263,148.462
C01359=1196.763,371.769,-78.170,-176.003,8.266,148.463
C01360=1196.759,372.016,-78.204,-176.002,8.269,148.463
C01361=1196.756,372.264,-78.238,-176.000,8.273,148.463
C01362=1196.751,372.512,-78.272,-175.999,8.276,148.464
C01363=1196.747,372.759,-78.306,-175.998,8.279,148.464
C01364=1196.743,373.007,-78.341,-175.996,8.282,148.465
C01365=1196.740,373.254,-78.375,-175.995,8.285,148.465
C01366=1196.735,373.502,-78.409,-175.993,8.289,148.466
C01367=1196.732,373.750,-78.443,-175.992,8.291,148.466
C01368=1196.727,373.997,-78.477,-175.991,8.295,148.467
C01369=1196.723,374.245,-78.511,-175.990,8.297,148.467
C01370=1196.719,374.493,-78.546,-175.988,8.301,148.467
C01371=1196.715,374.740,-78.579,-175.988,8.304,148.468
C01372=1196.711,374.989,-78.614,-175.986,8.307,148.468
C01373=1196.707,375.236,-78.648,-175.985,8.311,148.469
C01374=1196.703,375.483,-78.682,-175.984,8.314,148.469
C01375=1196.699,375.731,-78.717,-175.983,8.316,148.470
C01376=1196.695,375.978,-78.751,-175.981,8.319,148.470
C01377=1196.690,376.226,-78.785,-175.980,8.323,148.471
C01378=1196.687,376.474,-78.820,-175.979,8.326,148.471
C01379=1196.683,376.721,-78.854,-175.978,8.329,148.472
C01380=1196.679,376.969,-78.888,-175.977,8.332,148.472
C01381=1196.675,377.216,-78.923,-175.975,8.336,148.473
C01382=1196.670,377.464,-78.957,-175.974,8.339,148.473
C01383=1196.667,377.712,-78.991,-175.973,8.341,148.474
C01384=1196.662,377.959,-79.025,-175.972,8.344,148.474
C01385=1196.659,378.207,-79.060,-175.971,8.347,148.475
C01386=1196.654,378.455,-79.094,-175.970,8.350,148.475
C01387=1196.650,378.702,-79.128,-175.968,8.354,148.476
C01388=1196.646,378.950,-79.163,-175.967,8.357,148.476
C01389=1196.642,379.197,-79.197,-175.966,8.360,148.477
C01390=1196.639,379.445,-79.231,-175.965,8.363,148.477
C01391=1196.634,379.692,-79.267,-175.964,8.366,148.478
C01392=1196.630,379.940,-79.301,-175.964,8.369,148.478
C01393=1196.627,380.187,-79.335,-175.962,8.372,148.479
C01394=1196.622,380.435,-79.370,-175.962,8.375,148.479
C01395=1196.618,380.683,-79.405,-175.960,8.378,148.480
C01396=1196.614,380.930,-79.438,-175.960,8.381,148.480
C01397=1196.610,381.178,-79.473,-175.958,8.384,148.481
C01398=1196.606,381.425,-79.508,-175.957,8.388,148.481
C01399=1196.602,381.673,-79.542,-175.956,8.391,148.482
C01400=1196.598,381.921,-79.576,-175.955,8.393,148.482
C01401=1196.594,382.169,-79.611,-175.954,8.397,148.483
C01402=1196.589,382.416,-79.646,-175.953,8.400,148.483
C01403=1196.586,382.663,-79.681,-175.952,8.402,148.484
C01404=1196.582,382.911,-79.715,-175.951,8.406,148.484
C01405=1196.577,383.158,-79.750,-175.951,8.408,148.485
C01406=1196.574,383.406,-79.784,-175.950,8.411,148.485
C01407=1196.569,383.653,-79.818,-175.949,8.414,148.486
C01408=1196.565,383.902,-79.853,-175.948,8.417,148.486
C01409=1196.561,384.148,-79.888,-175.947,8.420,148.487
C01410=1196.558,384.396,-79.923,-175.946,8.423,148.487
C01411=1196.553,384.644,-79.957,-175.946,8.426,148.488
C01412=1196.549,384.892,-79.992,-175.945,8.429,148.489
C01413=1196.545,385.139,-80.026,-175.944,8.432,148.489
C01414=1196.542,385.386,-80.061,-175.943,8.435,148.490
C01415=1196.537,385.634,-80.096,-175.943,8.437,148.490
C01416=1196.533,385.882,-80.131,-175.942,8.440,148.491
C01417=1196.529,386.129,-80.165,-175.941,8.443,148.491
C01418=1196.526,386.376,-80.200,-175.940,8.446,148.492
C01419=1196.521,386.624,-80.235,-175.939,8.449,148.492
C01420=1196.517,386.872,-80.269,-175.939,8.451,148.493
C01421=1196.513,387.119,-80.305,-175.938,8.455,148.493
C01422=1196.509,387.367,-80.339,-175.937,8.458,148.494
C01423=1196.505,387.614,-80.373,-175.936,8.461,148.495
C01424=1196.501,387.862,-80.408,-175.936,8.463,148.495
C01425=1196.498,388.110,-80.444,-175.935,8.466,148.495
C01426=1196.493,388.357,-80.478,-175.934,8.469,148.496
C01427=1196.489,388.605,-80.513,-175.933,8.472,148.497
C01428=1196.486,388.852,-80.548,-175.933,8.474,148.497
C01429=1196.482,389.100,-80.582,-175.932,8.477,148.498
C01430=1196.477,389.347,-80.617,-175.932,8.481,148.498
C01431=1196.473,389.595,-80.652,-175.931,8.483,148.499
C01432=1196.469,389.842,-80.687,-175.931,8.486,148.499
C01433=1196.465,390.090,-80.722,-175.930,8.488,148.500
C01434=1196.461,390.337,-80.756,-175.930,8.491,148.501
C01435=1196.457,390.585,-80.791,-175.928,8.494,148.501
C01436=1196.454,390.832,-80.827,-175.928,8.496,148.502
C01437=1196.449,391.080,-80.861,-175.927,8.499,148.502
C01438=1196.445,391.328,-80.896,-175.927,8.502,148.503
C01439=1196.441,391.575,-80.931,-175.926,8.505,148.503
C01440=1196.437,391.823,-80.966,-175.926,8.508,148.504
C01441=1196.433,392.105,-81.006,-175.925,8.510,148.504
C01442=1196.428,392.389,-81.046,-175.925,8.514,148.505
C01443=1196.424,392.672,-81.086,-175.924,8.517,148.506
C01444=1196.418,392.955,-81.125,-175.923,8.520,148.506
C01445=1196.415,393.202,-81.161,-175.923,8.523,148.507
C01446=1196.411,393.450,-81.195,-175.922,8.525,148.507
C01447=1196.407,393.697,-81.230,-175.922,8.527,148.508
C01448=1196.403,393.945,-81.265,-175.921,8.531,148.509
C01449=1196.399,394.192,-81.300,-175.921,8.533,148.509
C01450=1196.395,394.440,-81.335,-175.920,8.536,148.510
C01451=1196.391,394.687,-81.371,-175.920,8.538,148.510
C01452=1196.387,394.935,-81.405,-175.919,8.541,148.511
C01453=1196.383,395.182,-81.441,-175.919,8.544,148.511
C01454=1196.379,395.430,-81.475,-175.919,8.546,148.512
C01455=1196.375,395.677,-81.511,-175.918,8.549,148.512
C01456=1196.371,395.925,-81.546,-175.918,8.551,148.513
C01457=1196.367,396.172,-81.581,-175.917,8.554,148.514
C01458=1196.363,396.420,-81.616,-175.917,8.557,148.514
C01459=1196.358,396.667,-81.651,-175.917,8.559,148.515
C01460=1196.354,396.915,-81.686,-175.916,8.562,148.515
C01461=1196.351,397.162,-81.721,-175.916,8.564,148.516
C01462=1196.347,397.409,-81.756,-175.915,8.566,148.516
C01463=1196.343,397.657,-81.791,-175.915,8.570,148.517
C01464=1196.340,397.905,-81.826,-175.914,8.572,148.517
C01465=1196.335,398.152,-81.861,-175.914,8.574,148.518
C01466=1196.331,398.400,-81.896,-175.914,8.577,148.519
C01467=1196.327,398.647,-81.931,-175.913,8.580,148.519
C01468=1196.323,398.895,-81.966,-175.913,8.582,148.520
C01469=1196.319,399.142,-82.002,-175.913,8.584,148.520
C01470=1196.315,399.390,-82.036,-175.913,8.587,148.521
C01471=1196.311,399.637,-82.072,-175.912,8.590,148.521
C01472=1196.307,399.885,-82.107,-175.912,8.592,148.522
C01473=1196.303,400.132,-82.142,-175.911,8.594,148.522
C01474=1196.299,400.380,-82.177,-175.911,8.596,148.523
C01475=1196.295,400.628,-82.212,-175.911,8.599,148.524
C01476=1196.291,400.874,-82.247,-175.910,8.602,148.524
C01477=1196.287,401.122,-82.283,-175.910,8.604,148.525
C01478=1196.283,401.369,-82.317,-175.910,8.606,148.525
C01479=1196.279,401.617,-82.353,-175.910,8.609,148.526
C01480=1196.276,401.864,-82.388,-175.909,8.611,148.526
C01481=1196.270,402.112,-82.423,-175.909,8.613,148.527
C01482=1196.267,402.360,-82.459,-175.908,8.616,148.527
C01483=1196.263,402.607,-82.495,-175.908,8.619,148.528
C01484=1196.258,402.855,-82.529,-175.908,8.621,148.528
C01485=1196.255,403.102,-82.565,-175.908,8.623,148.529
C01486=1196.251,403.350,-82.600,-175.907,8.625,148.529
C01487=1196.246,403.597,-82.635,-175.907,8.628,148.530
C01488=1196.243,403.844,-82.670,-175.907,8.630,148.531
C01489=1196.239,404.092,-82.706,-175.907,8.632,148.531
C01490=1196.235,404.339,-82.741,-175.906,8.634,148.532
C01491=1196.231,404.587,-82.776,-175.906,8.637,148.532
C01492=1196.227,404.834,-82.811,-175.905,8.640,148.533
C01493=1196.224,405.082,-82.847,-175.905,8.642,148.533
C01494=1196.219,405.329,-82.881,-175.905,8.644,148.534
C01495=1196.215,405.577,-82.917,-175.905,8.647,148.534
C01496=1196.212,405.824,-82.952,-175.904,8.649,148.535
C01497=1196.207,406.071,-82.988,-175.904,8.651,148.535
C01498=1196.203,406.320,-83.023,-175.904,8.653,148.536
C01499=1196.199,406.567,-83.059,-175.904,8.656,148.536
C01500=1196.195,406.814,-83.094,-175.903,8.658,148.537
C01501=1196.191,407.061,-83.129,-175.903,8.660,148.537
C01502=1196.187,407.309,-83.164,-175.903,8.662,148.538
C01503=1196.183,407.556,-83.199,-175.903,8.665,148.538
C01504=1196.179,407.804,-83.235,-175.903,8.667,148.539
C01505=1196.176,408.051,-83.270,-175.902,8.669,148.540
C01506=1196.172,408.299,-83.306,-175.902,8.671,148.540
C01507=1196.167,408.546,-83.340,-175.902,8.674,148.541
C01508=1196.163,408.794,-83.376,-175.902,8.675,148.541
C01509=1196.159,409.041,-83.412,-175.902,8.677,148.542
C01510=1196.155,409.288,-83.447,-175.902,8.680,148.542
C01511=1196.151,409.536,-83.483,-175.901,8.682,148.543
C01512=1196.147,409.784,-83.518,-175.901,8.684,148.543
C01513=1196.144,410.031,-83.553,-175.901,8.687,148.544
C01514=1196.139,410.278,-83.588,-175.901,8.689,148.544
C01515=1196.136,410.526,-83.624,-175.900,8.691,148.545
C01516=1196.131,410.774,-83.660,-175.900,8.693,148.545
C01517=1196.127,411.020,-83.695,-175.900,8.696,148.546
C01518=1196.123,411.268,-83.731,-175.900,8.698,148.546
C01519=1196.119,411.516,-83.766,-175.900,8.699,148.547
C01520=1196.116,411.763,-83.801,-175.900,8.702,148.547
C01521=1196.112,412.010,-83.836,-175.900,8.704,148.548
C01522=1196.108,412.258,-83.872,-175.899,8.706,148.548
C01523=1196.103,412.506,-83.908,-175.899,8.708,148.549
C01524=1196.100,412.753,-83.944,-175.898,8.710,148.549
C01525=1196.096,413.000,-83.979,-175.898,8.713,148.550
C01526=1196.092,413.248,-84.014,-175.898,8.714,148.550
C01527=1196.088,413.495,-84.049,-175.898,8.716,148.551
C01528=1196.084,413.743,-84.085,-175.898,8.719,148.551
C01529=1196.079,413.990,-84.120,-175.898,8.721,148.552
C01530=1196.076,414.238,-84.156,-175.898,8.723,148.552
C01531=1196.072,414.485,-84.192,-175.897,8.725,148.553
C01532=1196.068,414.733,-84.227,-175.898,8.727,148.553
C01533=1196.064,414.979,-84.262,-175.897,8.729,148.554
C01534=1196.060,415.227,-84.298,-175.897,8.731,148.554
C01535=1196.056,415.475,-84.334,-175.896,8.733,148.555
C01536=1196.052,415.722,-84.370,-175.897,8.735,148.555
C01537=1196.046,416.069,-84.419,-175.896,8.738,148.556
C01538=1196.043,416.415,-84.469,-175.896,8.740,148.557
C01539=1196.042,416.762,-84.517,-175.896,8.744,148.557
C01540=1196.044,417.108,-84.567,-175.896,8.746,148.558
C01541=1195.623,417.109,-84.606,-175.899,8.757,148.561
C01542=1195.620,416.759,-84.556,-175.899,8.754,148.561
C01543=1195.621,416.410,-84.507,-175.899,8.751,148.560
C01544=1195.625,416.061,-84.457,-175.900,8.749,148.560
C01545=1195.631,415.711,-84.407,-175.899,8.746,148.559
C01546=1195.635,415.463,-84.371,-175.900,8.744,148.558
C01547=1195.639,415.217,-84.336,-175.900,8.742,148.558
C01548=1195.642,414.969,-84.300,-175.900,8.740,148.558
C01549=1195.646,414.722,-84.265,-175.901,8.737,148.557
C01550=1195.650,414.474,-84.229,-175.900,8.736,148.557
C01551=1195.655,414.227,-84.193,-175.901,8.734,148.556
C01552=1195.658,413.979,-84.158,-175.901,8.731,148.555
C01553=1195.662,413.732,-84.122,-175.901,8.729,148.555
C01554=1195.666,413.484,-84.087,-175.901,8.727,148.554
C01555=1195.670,413.237,-84.052,-175.902,8.725,148.554
C01556=1195.675,412.989,-84.016,-175.901,8.723,148.553
C01557=1195.678,412.742,-83.981,-175.902,8.721,148.553
C01558=1195.682,412.494,-83.945,-175.902,8.719,148.552
C01559=1195.686,412.247,-83.910,-175.902,8.716,148.552
C01560=1195.690,412.000,-83.874,-175.903,8.714,148.552
C01561=1195.694,411.752,-83.839,-175.903,8.712,148.551
C01562=1195.698,411.505,-83.803,-175.903,8.711,148.551
C01563=1195.703,411.257,-83.768,-175.903,8.709,148.550
C01564=1195.706,411.010,-83.733,-175.903,8.706,148.549
C01565=1195.710,410.762,-83.697,-175.903,8.704,148.549
C01566=1195.714,410.515,-83.662,-175.904,8.702,148.548
C01567=1195.718,410.268,-83.626,-175.904,8.699,148.548
C01568=1195.722,410.020,-83.591,-175.904,8.697,148.547
C01569=1195.726,409.773,-83.555,-175.904,8.695,148.547
C01570=1195.730,409.525,-83.520,-175.905,8.693,148.546
C01571=1195.734,409.278,-83.485,-175.905,8.690,148.546
C01572=1195.738,409.030,-83.449,-175.904,8.689,148.545
C01573=1195.741,408.783,-83.414,-175.905,8.687,148.545
C01574=1195.746,408.536,-83.378,-175.905,8.684,148.544
C01575=1195.750,408.288,-83.344,-175.905,8.682,148.544
C01576=1195.753,408.040,-83.308,-175.905,8.680,148.543
C01577=1195.758,407.793,-83.272,-175.906,8.678,148.543
C01578=1195.762,407.546,-83.237,-175.906,8.675,148.542
C01579=1195.766,407.298,-83.201,-175.906,8.673,148.542
C01580=1195.770,407.050,-83.166,-175.906,8.671,148.541
C01581=1195.774,406.803,-83.131,-175.907,8.669,148.541
C01582=1195.778,406.556,-83.096,-175.907,8.666,148.540
C01583=1195.781,406.308,-83.060,-175.907,8.664,148.540
C01584=1195.786,406.061,-83.025,-175.907,8.662,148.539
C01585=1195.789,405.813,-82.990,-175.908,8.659,148.538
C01586=1195.793,405.566,-82.954,-175.908,8.657,148.538
C01587=1195.797,405.319,-82.919,-175.908,8.655,148.537
C01588=1195.802,405.071,-82.883,-175.908,8.653,148.537
C01589=1195.806,404.823,-82.848,-175.909,8.650,148.536
C01590=1195.810,404.576,-82.813,-175.909,8.648,148.536
C01591=1195.814,404.329,-82.778,-175.909,8.646,148.535
C01592=1195.818,404.081,-82.743,-175.909,8.644,148.535
C01593=1195.821,403.833,-82.707,-175.909,8.641,148.534
C01594=1195.826,403.586,-82.672,-175.910,8.638,148.534
C01595=1195.829,403.339,-82.636,-175.911,8.636,148.533
C01596=1195.833,403.091,-82.602,-175.911,8.634,148.533
C01597=1195.837,402.844,-82.566,-175.911,8.631,148.532
C01598=1195.841,402.596,-82.531,-175.911,8.629,148.532
C01599=1195.845,402.348,-82.496,-175.911,8.627,148.531
C01600=1195.849,402.101,-82.461,-175.911,8.624,148.530
C01601=1195.853,401.854,-82.425,-175.911,8.622,148.530
C01602=1195.857,401.606,-82.391,-175.912,8.620,148.529
C01603=1195.861,401.359,-82.355,-175.913,8.617,148.529
C01604=1195.865,401.112,-82.320,-175.913,8.614,148.528
C01605=1195.869,400.863,-82.285,-175.913,8.612,148.528
C01606=1195.873,400.617,-82.250,-175.913,8.610,148.527
C01607=1195.877,400.369,-82.214,-175.913,8.608,148.527
C01608=1195.881,400.122,-82.180,-175.914,8.605,148.526
C01609=1195.885,399.874,-82.144,-175.914,8.602,148.525
C01610=1195.889,399.627,-82.109,-175.915,8.600,148.525
C01611=1195.894,399.379,-82.074,-175.915,8.598,148.524
C01612=1195.898,399.131,-82.038,-175.915,8.595,148.524
C01613=1195.902,398.883,-82.003,-175.916,8.592,148.523
C01614=1195.906,398.637,-81.968,-175.916,8.590,148.523
C01615=1195.909,398.389,-81.933,-175.916,8.588,148.522
C01616=1195.913,398.141,-81.898,-175.917,8.586,148.522
C01617=1195.917,397.894,-81.863,-175.917,8.582,148.521
C01618=1195.921,397.646,-81.828,-175.918,8.580,148.521
C01619=1195.925,397.400,-81.793,-175.918,8.578,148.520
C01620=1195.929,397.152,-81.758,-175.919,8.575,148.519
C01621=1195.933,396.904,-81.723,-175.919,8.573,148.519
C01622=1195.937,396.657,-81.687,-175.919,8.570,148.518
C01623=1195.941,396.409,-81.653,-175.920,8.567,148.518
C01624=1195.945,396.161,-81.617,-175.920,8.565,148.517
C01625=1195.949,395.914,-81.583,-175.920,8.562,148.517
C01626=1195.953,395.667,-81.547,-175.921,8.559,148.516
C01627=1195.958,395.419,-81.513,-175.921,8.557,148.515
C01628=1195.961,395.172,-81.477,-175.921,8.555,148.515
C01629=1195.965,394.923,-81.442,-175.922,8.552,148.514
C01630=1195.970,394.677,-81.407,-175.922,8.549,148.514
C01631=1195.974,394.429,-81.372,-175.923,8.546,148.513
C01632=1195.978,394.182,-81.337,-175.923,8.544,148.513
C01633=1195.982,393.934,-81.302,-175.924,8.541,148.512
C01634=1195.985,393.686,-81.267,-175.924,8.539,148.512
C01635=1195.990,393.439,-81.232,-175.925,8.536,148.511
C01636=1195.993,393.192,-81.197,-175.925,8.533,148.510
C01637=1195.997,392.944,-81.163,-175.926,8.531,148.510
C01638=1196.002,392.661,-81.122,-175.926,8.528,148.509
C01639=1196.006,392.378,-81.083,-175.927,8.525,148.509
C01640=1196.011,392.094,-81.042,-175.928,8.521,148.508
C01641=1196.016,391.812,-81.002,-175.928,8.518,148.507
C01642=1196.019,391.564,-80.967,-175.929,8.515,148.507
C01643=1196.024,391.317,-80.933,-175.929,8.513,148.506
C01644=1196.027,391.069,-80.897,-175.930,8.510,148.506
C01645=1196.032,390.822,-80.863,-175.930,8.508,148.505
C01646=1196.036,390.574,-80.827,-175.931,8.504,148.504
C01647=1196.040,390.326,-80.793,-175.931,8.502,148.504
C01648=1196.044,390.079,-80.758,-175.932,8.499,148.503
C01649=1196.047,389.831,-80.723,-175.933,8.496,148.503
C01650=1196.052,389.584,-80.689,-175.934,8.494,148.502
C01651=1196.055,389.336,-80.653,-175.934,8.491,148.502
C01652=1196.060,389.089,-80.619,-175.935,8.488,148.501
C01653=1196.064,388.841,-80.584,-175.935,8.486,148.501
C01654=1196.068,388.594,-80.549,-175.936,8.482,148.500
C01655=1196.071,388.346,-80.514,-175.937,8.479,148.500
C01656=1196.076,388.099,-80.480,-175.937,8.477,148.499
C01657=1196.080,387.851,-80.444,-175.938,8.474,148.498
C01658=1196.084,387.603,-80.410,-175.939,8.471,148.498
C01659=1196.088,387.356,-80.375,-175.940,8.468,148.497
C01660=1196.091,387.109,-80.340,-175.940,8.466,148.497
C01661=1196.096,386.861,-80.306,-175.941,8.463,148.496
C01662=1196.100,386.613,-80.271,-175.942,8.460,148.496
C01663=1196.104,386.366,-80.236,-175.943,8.456,148.495
C01664=1196.108,386.118,-80.201,-175.943,8.454,148.495
C01665=1196.112,385.871,-80.167,-175.944,8.451,148.494
C01666=1196.116,385.623,-80.132,-175.945,8.448,148.494
C01667=1196.120,385.376,-80.098,-175.946,8.445,148.493
C01668=1196.124,385.128,-80.062,-175.946,8.442,148.492
C01669=1196.128,384.881,-80.028,-175.947,8.439,148.492
C01670=1196.132,384.633,-79.993,-175.948,8.436,148.492
C01671=1196.136,384.385,-79.959,-175.949,8.434,148.491
C01672=1196.140,384.138,-79.923,-175.949,8.431,148.490
C01673=1196.144,383.890,-79.889,-175.950,8.428,148.490
C01674=1196.148,383.643,-79.855,-175.951,8.425,148.489
C01675=1196.152,383.395,-79.820,-175.952,8.422,148.489
C01676=1196.156,383.147,-79.785,-175.953,8.419,148.488
C01677=1196.160,382.901,-79.751,-175.954,8.416,148.488
C01678=1196.164,382.653,-79.716,-175.955,8.413,148.487
C01679=1196.168,382.405,-79.682,-175.956,8.410,148.487
C01680=1196.172,382.157,-79.647,-175.957,8.407,148.486
C01681=1196.176,381.910,-79.613,-175.958,8.404,148.486
C01682=1196.181,381.662,-79.578,-175.959,8.401,148.485
C01683=1196.185,381.414,-79.544,-175.959,8.398,148.485
C01684=1196.188,381.167,-79.510,-175.961,8.395,148.484
C01685=1196.192,380.920,-79.474,-175.961,8.392,148.484
C01686=1196.197,380.672,-79.440,-175.963,8.389,148.483
C01687=1196.200,380.424,-79.405,-175.963,8.386,148.483
C01688=1196.204,380.177,-79.371,-175.964,8.383,148.482
C01689=1196.208,379.929,-79.336,-175.965,8.380,148.482
C01690=1196.212,379.682,-79.302,-175.967,8.376,148.481
C01691=1196.217,379.434,-79.268,-175.968,8.373,148.481
C01692=1196.221,379.186,-79.233,-175.969,8.370,148.480
C01693=1196.225,378.939,-79.199,-175.970,8.367,148.480
C01694=1196.229,378.691,-79.164,-175.971,8.364,148.479
C01695=1196.233,378.444,-79.130,-175.972,8.361,148.479
C01696=1196.236,378.196,-79.096,-175.973,8.358,148.478
C01697=1196.241,377.948,-79.061,-175.975,8.355,148.478
C01698=1196.245,377.701,-79.027,-175.975,8.352,148.477
C01699=1196.249,377.453,-78.992,-175.977,8.349,148.477
C01700=1196.253,377.206,-78.958,-175.977,8.346,148.476
C01701=1196.257,376.958,-78.924,-175.979,8.343,148.476
C01702=1196.261,376.711,-78.889,-175.980,8.339,148.475
C01703=1196.265,376.463,-78.855,-175.981,8.336,148.475
C01704=1196.269,376.215,-78.821,-175.982,8.333,148.474
C01705=1196.274,375.968,-78.786,-175.983,8.330,148.474
C01706=1196.277,375.720,-78.752,-175.985,8.327,148.473
C01707=1196.281,375.473,-78.717,-175.986,8.324,148.473
C01708=1196.285,375.225,-78.684,-175.987,8.321,148.472
C01709=1196.289,374.977,-78.649,-175.988,8.318,148.472
C01710=1196.293,374.730,-78.615,-175.990,8.314,148.471
C01711=1196.298,374.482,-78.581,-175.991,8.311,148.471
C01712=1196.301,374.234,-78.547,-175.992,8.308,148.470
C01713=1196.306,373.987,-78.512,-175.994,8.305,148.470
C01714=1196.309,373.739,-78.478,-175.995,8.302,148.470
C01715=1196.314,373.491,-78.444,-175.996,8.299,148.469
C01716=1196.318,373.244,-78.410,-175.998,8.295,148.469
C01717=1196.322,372.996,-78.376,-175.999,8.292,148.468
C01718=1196.325,372.749,-78.342,-176.000,8.290,148.468
C01719=1196.330,372.501,-78.307,-176.002,8.286,148.467
C01720=1196.334,372.253,-78.274,-176.003,8.283,148.467
C01721=1196.338,372.006,-78.239,-176.004,8.280,148.466
C01722=1196.342,371.758,-78.205,-176.006,8.276,148.466
C01723=1196.346,371.510,-78.171,-176.007,8.274,148.466
C01724=1196.350,371.263,-78.137,-176.009,8.270,148.465
C01725=1196.355,371.015,-78.103,-176.010,8.267,148.465
C01726=1196.358,370.767,-78.069,-176.011,8.264,148.464
C01727=1196.362,370.520,-78.035,-176.012,8.260,148.464
C01728=1196.367,370.272,-78.001,-176.014,8.258,148.463
C01729=1196.370,370.024,-77.967,-176.015,8.254,148.463
C01730=1196.374,369.777,-77.932,-176.017,8.251,148.462
C01731=1196.378,369.529,-77.899,-176.018,8.248,148.462
C01732=1196.382,369.282,-77.865,-176.020,8.245,148.462
C01733=1196.386,369.034,-77.831,-176.022,8.241,148.461
C01734=1196.390,368.786,-77.797,-176.023,8.238,148.461
C01735=1196.395,368.539,-77.763,-176.025,8.235,148.460
C01736=1196.399,368.291,-77.730,-176.026,8.232,148.460
C01737=1196.402,368.043,-77.696,-176.028,8.228,148.460
C01738=1196.407,367.796,-77.661,-176.029,8.225,148.459
C01739=1196.411,367.548,-77.628,-176.031,8.222,148.459
C01740=1196.414,367.300,-77.594,-176.032,8.219,148.458
C01741=1196.419,367.052,-77.560,-176.034,8.215,148.458
C01742=1196.424,366.772,-77.521,-176.035,8.212,148.457
C01743=1196.429,366.491,-77.483,-176.037,8.208,148.457
C01744=1196.433,366.211,-77.445,-176.039,8.204,148.457
C01745=1196.437,365.929,-77.407,-176.041,8.201,148.456
C01746=1196.442,365.681,-77.372,-176.042,8.198,148.456
C01747=1196.446,365.434,-77.339,-176.044,8.195,148.456
C01748=1196.450,365.187,-77.305,-176.046,8.191,148.455
C01749=1196.453,364.938,-77.272,-176.047,8.188,148.455
C01750=1196.458,364.691,-77.237,-176.049,8.185,148.454
C01751=1196.462,364.443,-77.204,-176.051,8.182,148.454
C01752=1196.466,364.196,-77.170,-176.052,8.178,148.454
C01753=1196.470,363.948,-77.137,-176.054,8.175,148.453
C01754=1196.474,363.700,-77.102,-176.055,8.172,148.453
C01755=1196.478,363.452,-77.069,-176.058,8.169,148.453
C01756=1196.482,363.205,-77.036,-176.059,8.166,148.452
C01757=1196.486,362.958,-77.002,-176.061,8.162,148.452
C01758=1196.491,362.710,-76.968,-176.063,8.159,148.452
C01759=1196.494,362.462,-76.934,-176.064,8.156,148.451
C01760=1196.498,362.214,-76.901,-176.066,8.152,148.451
C01761=1196.502,361.966,-76.868,-176.068,8.149,148.451
C01762=1196.506,361.719,-76.834,-176.069,8.146,148.450
C01763=1196.510,361.471,-76.801,-176.071,8.143,148.450
C01764=1196.515,361.223,-76.767,-176.073,8.139,148.449
C01765=1196.519,360.975,-76.734,-176.075,8.137,148.449
C01766=1196.523,360.728,-76.700,-176.076,8.133,148.449
C01767=1196.527,360.480,-76.667,-176.079,8.130,148.448
C01768=1196.531,360.232,-76.633,-176.080,8.127,148.448
C01769=1196.535,359.985,-76.600,-176.082,8.123,148.448
C01770=1196.539,359.737,-76.566,-176.084,8.120,148.447
C01771=1196.543,359.489,-76.532,-176.085,8.117,148.447
C01772=1196.547,359.241,-76.499,-176.087,8.114,148.447
C01773=1196.551,358.993,-76.466,-176.090,8.110,148.447
C01774=1196.555,358.746,-76.432,-176.091,8.107,148.446
C01775=1196.559,358.498,-76.399,-176.093,8.104,148.446
C01776=1196.563,358.251,-76.366,-176.095,8.101,148.445
C01777=1196.568,358.003,-76.333,-176.097,8.097,148.445
C01778=1196.572,357.755,-76.299,-176.098,8.094,148.445
C01779=1196.576,357.508,-76.266,-176.100,8.091,148.445
C01780=1196.579,357.259,-76.233,-176.102,8.087,148.444
C01781=1196.583,357.012,-76.199,-176.104,8.084,148.444
C01782=1196.588,356.764,-76.165,-176.106,8.082,148.444
C01783=1196.592,356.516,-76.132,-176.108,8.078,148.443
C01784=1196.596,356.269,-76.099,-176.110,8.075,148.443
C01785=1196.600,356.021,-76.066,-176.112,8.071,148.443
C01786=1196.605,355.773,-76.033,-176.114,8.069,148.443
C01787=1196.609,355.525,-75.999,-176.116,8.065,148.442
C01788=1196.613,355.278,-75.966,-176.118,8.062,148.442
C01789=1196.617,355.030,-75.933,-176.120,8.058,148.442
C01790=1196.621,354.782,-75.900,-176.122,8.056,148.441
C01791=1196.625,354.534,-75.867,-176.123,8.052,148.441
C01792=1196.629,354.287,-75.834,-176.126,8.049,148.441
C01793=1196.634,354.039,-75.800,-176.127,8.046,148.441
C01794=1196.637,353.792,-75.768,-176.129,8.043,148.440
C01795=1196.641,353.544,-75.735,-176.131,8.039,148.440
C01796=1196.645,353.296,-75.702,-176.133,8.036,148.440
C01797=1196.649,353.048,-75.668,-176.135,8.033,148.440
C01798=1196.654,352.800,-75.636,-176.137,8.030,148.439
C01799=1196.658,352.552,-75.603,-176.139,8.026,148.439
C01800=1196.662,352.305,-75.570,-176.141,8.023,148.439
C01801=1196.666,352.057,-75.537,-176.143,8.021,148.438
C01802=1196.670,351.809,-75.503,-176.145,8.017,148.438
C01803=1196.675,351.561,-75.470,-176.147,8.014,148.438
C01804=1196.679,351.314,-75.437,-176.149,8.010,148.438
C01805=1196.683,351.065,-75.405,-176.151,8.008,148.437
C01806=1196.687,350.818,-75.372,-176.153,8.005,148.437
C01807=1196.691,350.570,-75.339,-176.155,8.001,148.437
C01808=1196.695,350.322,-75.306,-176.158,7.998,148.437
C01809=1196.699,350.075,-75.273,-176.159,7.995,148.436
C01810=1196.703,349.826,-75.240,-176.161,7.992,148.436
C01811=1196.708,349.579,-75.207,-176.163,7.988,148.436
C01812=1196.711,349.331,-75.174,-176.166,7.985,148.436
C01813=1196.715,349.083,-75.141,-176.167,7.983,148.436
C01814=1196.719,348.835,-75.109,-176.169,7.979,148.435
